LIN {X 0,Y 471.276,Z 351.121,A -85,B 0,C 180,E1 -7520.71,E2 -7520.71} C_VEL
LIN {X 0,Y 472.038,Z 338.499,A -85,B 0,C 180,E1 -7521.712,E2 -7521.712} C_VEL
LIN {X 0,Y 472.825,Z 324.903,A -85,B 0,C 180,E1 -7522.589,E2 -7522.589} C_VEL
LIN {X 0,Y 473.432,Z 311.439,A -85,B 0,C 180,E1 -7523.284,E2 -7523.284} C_VEL
LIN {X 0,Y 473.938,Z 296.086,A -85,B 0,C 180,E1 -7523.884,E2 -7523.884} C_VEL
LIN {X 0,Y 469.116,Z 281.186,A -85,B 0,C 180,E1 -7524.542,E2 -7524.542} C_VEL
LIN {X 0,Y 466.998,Z 274.89,A -85,B 0,C 180,E1 -7524.795,E2 -7524.795} C_VEL
LIN {X 0,Y 467.098,Z 272.572,A -85,B 0,C 180,E1 -7527.412,E2 -7527.412} C_VEL
LIN {X 0,Y 467.145,Z 270.085,A -85,B 0,C 180,E1 -7530.235,E2 -7530.235} C_VEL
LIN {X 0,Y 467.191,Z 267.524,A -85,B 0,C 180,E1 -7533.175,E2 -7533.175} C_VEL
LIN {X 0,Y 467.265,Z 265.036,A -85,B 0,C 180,E1 -7536.041,E2 -7536.041} C_VEL
LIN {X 0,Y 467.335,Z 262.608,A -85,B 0,C 180,E1 -7538.844,E2 -7538.844} C_VEL
LIN {X 0,Y 467.354,Z 261.899,A -85,B 0,C 180,E1 -7539.766,E2 -7539.766} C_VEL
LIN {X 0,Y 467.561,Z 261.875,A -85,B 0,C 180,E1 -7542.506,E2 -7542.506} C_VEL
LIN {X 0,Y 467.599,Z 261.867,A -85,B 0,C 180,E1 -7545.197,E2 -7545.197} C_VEL
LIN {X 0,Y 467.649,Z 261.86,A -85,B 0,C 180,E1 -7547.855,E2 -7547.855} C_VEL
LIN {X 0,Y 467.676,Z 261.856,A -85,B 0,C 180,E1 -7551.358,E2 -7551.358} C_VEL
LIN {X 0,Y 467.739,Z 261.849,A -85,B 0,C 180,E1 -7553.964,E2 -7553.964} C_VEL
LIN {X 0,Y 467.856,Z 261.833,A -85,B 0,C 180,E1 -7557.418,E2 -7557.418} C_VEL
LIN {X 0,Y 467.878,Z 261.829,A -85,B 0,C 180,E1 -7560.001,E2 -7560.001} C_VEL
LIN {X 0,Y 467.856,Z 261.835,A -85,B 0,C 180,E1 -7562.584,E2 -7562.584} C_VEL
LIN {X 0,Y 467.741,Z 261.846,A -85,B 0,C 180,E1 -7566.038,E2 -7566.038} C_VEL
LIN {X 0,Y 467.679,Z 261.855,A -85,B 0,C 180,E1 -7568.644,E2 -7568.644} C_VEL
LIN {X 0,Y 467.653,Z 261.859,A -85,B 0,C 180,E1 -7572.146,E2 -7572.146} C_VEL
LIN {X 0,Y 467.636,Z 261.86,A -85,B 0,C 180,E1 -7575.696,E2 -7575.696} C_VEL
LIN {X 0,Y 467.615,Z 261.863,A -85,B 0,C 180,E1 -7578.766,E2 -7578.766} C_VEL
LIN {X 0,Y 467.579,Z 261.868,A -85,B 0,C 180,E1 -7581.269,E2 -7581.269} C_VEL
LIN {X 0,Y 467.571,Z 261.869,A -85,B 0,C 180,E1 -7583.944,E2 -7583.944} C_VEL
LIN {X 0,Y 467.626,Z 261.863,A -85,B 0,C 180,E1 -7586.8,E2 -7586.8} C_VEL
LIN {X 0,Y 467.552,Z 261.875,A -85,B 0,C 180,E1 -7589.739,E2 -7589.739} C_VEL
LIN {X 0,Y 467.581,Z 261.872,A -85,B 0,C 180,E1 -7592.759,E2 -7592.759} C_VEL
LIN {X 0,Y 467.551,Z 261.878,A -85,B 0,C 180,E1 -7595.89,E2 -7595.89} C_VEL
LIN {X 0,Y 467.581,Z 261.871,A -85,B 0,C 180,E1 -7599.145,E2 -7599.145} C_VEL
LIN {X 0,Y 467.594,Z 262,A -85,B 0,C 180,E1 -7601.978,E2 -7601.978} C_VEL
LIN {X 0,Y 468.651,Z 267.711,A -85,B 0,C 180,E1 -7605.186,E2 -7605.186} C_VEL
LIN {X 0,Y 469.319,Z 271.579,A -85,B 0,C 180,E1 -7607.204,E2 -7607.204} C_VEL
LIN {X 0,Y 469.458,Z 275.977,A -85,B 0,C 180,E1 -7609.34,E2 -7609.34} C_VEL
LIN {X 0,Y 469.141,Z 282.253,A -85,B 0,C 180,E1 -7612.107,E2 -7612.107} C_VEL
LIN {X 0,Y 468.696,Z 290.547,A -85,B 0,C 180,E1 -7615.56,E2 -7615.56} C_VEL
LIN {X 0,Y 468.411,Z 297.548,A -85,B 0,C 180,E1 -7618.323,E2 -7618.323} C_VEL
LIN {X 0,Y 468.186,Z 305.313,A -85,B 0,C 180,E1 -7621.292,E2 -7621.292} C_VEL
LIN {X 0,Y 467.915,Z 313.672,A -85,B 0,C 180,E1 -7624.315,E2 -7624.315} C_VEL
LIN {X 0,Y 467.634,Z 322.474,A -85,B 0,C 180,E1 -7627.466,E2 -7627.466} C_VEL
LIN {X 0,Y 467.569,Z 324.53,A -85,B 0,C 180,E1 -7628.201,E2 -7628.201} C_VEL
LIN {X 0,Y 472.227,Z 343.185,A -85,B 0,C 180,E1 -7628.827,E2 -7628.827} C_VEL
LIN {X 0,Y 473.825,Z 350.535,A -85,B 0,C 180,E1 -7629.124,E2 -7629.124} C_VEL
LIN {X 0,Y 473.197,Z 365.272,A -85,B 0,C 180,E1 -7629.681,E2 -7629.681} C_VEL
LIN {X 0,Y 472.446,Z 380.48,A -85,B 0,C 180,E1 -7630.446,E2 -7630.446} C_VEL
LIN {X 0,Y 471.604,Z 394.063,A -85,B 0,C 180,E1 -7631.314,E2 -7631.314} C_VEL
LIN {X 0,Y 470.728,Z 407.908,A -85,B 0,C 180,E1 -7632.403,E2 -7632.403} C_VEL
LIN {X 0,Y 469.94,Z 420.362,A -85,B 0,C 180,E1 -7633.604,E2 -7633.604} C_VEL
LIN {X 0,Y 469.159,Z 430.752,A -85,B 0,C 180,E1 -7634.803,E2 -7634.803} C_VEL
LIN {X 0,Y 468.478,Z 440.392,A -85,B 0,C 180,E1 -7636.112,E2 -7636.112} C_VEL
LIN {X 0,Y 467.823,Z 449.354,A -85,B 0,C 180,E1 -7637.55,E2 -7637.55} C_VEL
LIN {X 0,Y 467.513,Z 457.737,A -85,B 0,C 180,E1 -7639.17,E2 -7639.17} C_VEL
LIN {X 0,Y 467.072,Z 465.091,A -85,B 0,C 180,E1 -7640.91,E2 -7640.91} C_VEL
LIN {X 0,Y 466.831,Z 470.922,A -85,B 0,C 180,E1 -7642.649,E2 -7642.649} C_VEL
LIN {X 0,Y 466.777,Z 474.387,A -85,B 0,C 180,E1 -7643.951,E2 -7643.951} C_VEL
LIN {X 0,Y 466.62,Z 477.888,A -85,B 0,C 180,E1 -7645.682,E2 -7645.682} C_VEL
LIN {X 0,Y 466.639,Z 480.189,A -85,B 0,C 180,E1 -7647.411,E2 -7647.411} C_VEL
LIN {X 0,Y 466.587,Z 481.348,A -85,B 0,C 180,E1 -7649.138,E2 -7649.138} C_VEL
LIN {X 0,Y 466.587,Z 481.347,A -85,B 0,C 180,E1 -7650.864,E2 -7650.864} C_VEL
LIN {X 0,Y 466.639,Z 480.185,A -85,B 0,C 180,E1 -7652.59,E2 -7652.59} C_VEL
LIN {X 0,Y 466.62,Z 477.881,A -85,B 0,C 180,E1 -7654.319,E2 -7654.319} C_VEL
LIN {X 0,Y 466.751,Z 474.385,A -85,B 0,C 180,E1 -7656.051,E2 -7656.051} C_VEL
LIN {X 0,Y 466.891,Z 469.607,A -85,B 0,C 180,E1 -7657.787,E2 -7657.787} C_VEL
LIN {X 0,Y 467.139,Z 463.417,A -85,B 0,C 180,E1 -7659.526,E2 -7659.526} C_VEL
LIN {X 0,Y 467.628,Z 455.639,A -85,B 0,C 180,E1 -7661.267,E2 -7661.267} C_VEL
LIN {X 0,Y 468.038,Z 447.109,A -85,B 0,C 180,E1 -7662.838,E2 -7662.838} C_VEL
LIN {X 0,Y 468.746,Z 437.387,A -85,B 0,C 180,E1 -7664.324,E2 -7664.324} C_VEL
LIN {X 0,Y 469.354,Z 427.179,A -85,B 0,C 180,E1 -7665.637,E2 -7665.637} C_VEL
LIN {X 0,Y 470.255,Z 414.818,A -85,B 0,C 180,E1 -7666.964,E2 -7666.964} C_VEL
LIN {X 0,Y 471.111,Z 401.347,A -85,B 0,C 180,E1 -7668.145,E2 -7668.145} C_VEL
LIN {X 0,Y 471.975,Z 387.646,A -85,B 0,C 180,E1 -7669.123,E2 -7669.123} C_VEL
LIN {X 0,Y 472.81,Z 373.473,A -85,B 0,C 180,E1 -7669.935,E2 -7669.935} C_VEL
LIN {X 0,Y 473.538,Z 357.964,A -85,B 0,C 180,E1 -7670.619,E2 -7670.619} C_VEL
LIN {X 0,Y 473.65,Z 349.449,A -85,B 0,C 180,E1 -7670.92,E2 -7670.92} C_VEL
LIN {X 0,Y 469.919,Z 334.013,A -85,B 0,C 180,E1 -7671.505,E2 -7671.505} C_VEL
LIN {X 0,Y 467.609,Z 324.753,A -85,B 0,C 180,E1 -7671.797,E2 -7671.797} C_VEL
LIN {X 0,Y 467.901,Z 315.127,A -85,B 0,C 180,E1 -7675.278,E2 -7675.278} C_VEL
LIN {X 0,Y 468.225,Z 305.789,A -85,B 0,C 180,E1 -7678.707,E2 -7678.707} C_VEL
LIN {X 0,Y 468.466,Z 298.067,A -85,B 0,C 180,E1 -7681.674,E2 -7681.674} C_VEL
LIN {X 0,Y 468.842,Z 290.541,A -85,B 0,C 180,E1 -7684.725,E2 -7684.725} C_VEL
LIN {X 0,Y 469.25,Z 282.979,A -85,B 0,C 180,E1 -7687.884,E2 -7687.884} C_VEL
LIN {X 0,Y 469.561,Z 276.677,A -85,B 0,C 180,E1 -7690.664,E2 -7690.664} C_VEL
LIN {X 0,Y 469.383,Z 272.101,A -85,B 0,C 180,E1 -7692.805,E2 -7692.805} C_VEL
LIN {X 0,Y 468.589,Z 267.36,A -85,B 0,C 180,E1 -7695.177,E2 -7695.177} C_VEL
LIN {X 0,Y 467.58,Z 261.869,A -85,B 0,C 180,E1 -7698.165,E2 -7698.165} C_VEL
LIN {X 0,Y 467.567,Z 261.87,A -85,B 0,C 180,E1 -7701.409,E2 -7701.409} C_VEL
LIN {X 0,Y 467.564,Z 261.869,A -85,B 0,C 180,E1 -7704.261,E2 -7704.261} C_VEL
LIN {X 0,Y 467.585,Z 261.867,A -85,B 0,C 180,E1 -7707.321,E2 -7707.321} C_VEL
LIN {X 0,Y 467.574,Z 261.869,A -85,B 0,C 180,E1 -7710.667,E2 -7710.667} C_VEL
LIN {X 0,Y 467.622,Z 261.862,A -85,B 0,C 180,E1 -7713.199,E2 -7713.199} C_VEL
LIN {X 0,Y 467.598,Z 261.867,A -85,B 0,C 180,E1 -7716.468,E2 -7716.468} C_VEL
LIN {X 0,Y 467.629,Z 261.859,A -85,B 0,C 180,E1 -7719.777,E2 -7719.777} C_VEL
LIN {X 0,Y 467.615,Z 261.865,A -85,B 0,C 180,E1 -7722.506,E2 -7722.506} C_VEL
LIN {X 0,Y 467.611,Z 261.864,A -85,B 0,C 180,E1 -7725.196,E2 -7725.196} C_VEL
LIN {X 0,Y 467.661,Z 261.857,A -85,B 0,C 180,E1 -7727.854,E2 -7727.854} C_VEL
LIN {X 0,Y 467.685,Z 261.853,A -85,B 0,C 180,E1 -7731.356,E2 -7731.356} C_VEL
LIN {X 0,Y 467.726,Z 261.849,A -85,B 0,C 180,E1 -7733.962,E2 -7733.962} C_VEL
LIN {X 0,Y 467.864,Z 261.83,A -85,B 0,C 180,E1 -7737.416,E2 -7737.416} C_VEL
LIN {X 0,Y 467.887,Z 261.829,A -85,B 0,C 180,E1 -7739.999,E2 -7739.999} C_VEL
LIN {X 0,Y 467.862,Z 261.833,A -85,B 0,C 180,E1 -7742.582,E2 -7742.582} C_VEL
LIN {X 0,Y 467.746,Z 261.847,A -85,B 0,C 180,E1 -7746.036,E2 -7746.036} C_VEL
LIN {X 0,Y 467.684,Z 261.855,A -85,B 0,C 180,E1 -7748.642,E2 -7748.642} C_VEL
LIN {X 0,Y 467.658,Z 261.859,A -85,B 0,C 180,E1 -7752.144,E2 -7752.144} C_VEL
LIN {X 0,Y 467.641,Z 261.859,A -85,B 0,C 180,E1 -7755.694,E2 -7755.694} C_VEL
LIN {X 0,Y 467.618,Z 261.863,A -85,B 0,C 180,E1 -7758.763,E2 -7758.763} C_VEL
LIN {X 0,Y 467.581,Z 261.866,A -85,B 0,C 180,E1 -7761.267,E2 -7761.267} C_VEL
LIN {X 0,Y 467.573,Z 261.869,A -85,B 0,C 180,E1 -7763.942,E2 -7763.942} C_VEL
LIN {X 0,Y 467.616,Z 261.862,A -85,B 0,C 180,E1 -7766.799,E2 -7766.799} C_VEL
LIN {X 0,Y 467.553,Z 261.873,A -85,B 0,C 180,E1 -7769.737,E2 -7769.737} C_VEL
LIN {X 0,Y 467.581,Z 261.866,A -85,B 0,C 180,E1 -7772.757,E2 -7772.757} C_VEL
LIN {X 0,Y 467.554,Z 261.873,A -85,B 0,C 180,E1 -7775.888,E2 -7775.888} C_VEL
LIN {X 0,Y 467.579,Z 261.867,A -85,B 0,C 180,E1 -7779.143,E2 -7779.143} C_VEL
LIN {X 0,Y 467.582,Z 261.867,A -85,B 0,C 180,E1 -7782.566,E2 -7782.566} C_VEL
LIN {X 0,Y 467.566,Z 261.868,A -85,B 0,C 180,E1 -7785.052,E2 -7785.052} C_VEL
LIN {X 0,Y 467.619,Z 261.864,A -85,B 0,C 180,E1 -7787.443,E2 -7787.443} C_VEL
LIN {X 0,Y 467.594,Z 261.864,A -85,B 0,C 180,E1 -7790.856,E2 -7790.856} C_VEL
LIN {X 0,Y 467.556,Z 261.871,A -85,B 0,C 180,E1 -7794.259,E2 -7794.259} C_VEL
LIN {X 0,Y 467.575,Z 261.869,A -85,B 0,C 180,E1 -7797.32,E2 -7797.32} C_VEL
LIN {X 0,Y 467.57,Z 261.867,A -85,B 0,C 180,E1 -7800.664,E2 -7800.664} C_VEL
LIN {X 0,Y 467.62,Z 261.864,A -85,B 0,C 180,E1 -7803.199,E2 -7803.199} C_VEL
LIN {X 0,Y 467.584,Z 261.865,A -85,B 0,C 180,E1 -7806.467,E2 -7806.467} C_VEL
LIN {X 0,Y 467.615,Z 261.864,A -85,B 0,C 180,E1 -7809.776,E2 -7809.776} C_VEL
LIN {X 0,Y 467.6,Z 261.864,A -85,B 0,C 180,E1 -7812.506,E2 -7812.506} C_VEL
LIN {X 0,Y 467.59,Z 261.866,A -85,B 0,C 180,E1 -7815.418,E2 -7815.418} C_VEL
LIN {X 0,Y 466.921,Z 261.949,A -85,B 0,C 180,E1 -7816.137,E2 -7816.137} C_VEL
LIN {X 0,Y 464.086,Z 262.304,A -85,B 0,C 180,E1 -7817.306,E2 -7817.306} C_VEL
LIN {X 0,Y 461.692,Z 262.599,A -85,B 0,C 180,E1 -7818.248,E2 -7818.248} C_VEL
LIN {X 0,Y 460.665,Z 262.73,A -85,B 0,C 180,E1 -7818.976,E2 -7818.976} C_VEL
LIN {X 0,Y 460.581,Z 262.739,A -85,B 0,C 180,E1 -7819.223,E2 -7819.223} C_VEL
LIN {X 0,Y 460.709,Z 262.721,A -85,B 0,C 180,E1 -7822.537,E2 -7822.537} C_VEL
LIN {X 0,Y 460.668,Z 262.727,A -85,B 0,C 180,E1 -7824.747,E2 -7824.747} C_VEL
LIN {X 0,Y 460.337,Z 262.772,A -85,B 0,C 180,E1 -7828.25,E2 -7828.25} C_VEL
LIN {X 0,Y 460.531,Z 263.298,A -85,B 0,C 180,E1 -7829.125,E2 -7829.125} C_VEL
LIN {X 0,Y 460.006,Z 265.723,A -85,B 0,C 180,E1 -7831.75,E2 -7831.75} C_VEL
LIN {X 0,Y 460.14,Z 268.114,A -85,B 0,C 180,E1 -7834.379,E2 -7834.379} C_VEL
LIN {X 0,Y 460.034,Z 270.553,A -85,B 0,C 180,E1 -7837.019,E2 -7837.019} C_VEL
LIN {X 0,Y 459.895,Z 273.884,A -85,B 0,C 180,E1 -7840.566,E2 -7840.566} C_VEL
LIN {X 0,Y 459.941,Z 274.351,A -85,B 0,C 180,E1 -7840.983,E2 -7840.983} C_VEL
LIN {X 0,Y 464.985,Z 289.981,A -85,B 0,C 180,E1 -7841.608,E2 -7841.608} C_VEL
LIN {X 0,Y 467.218,Z 298.137,A -85,B 0,C 180,E1 -7841.99,E2 -7841.99} C_VEL
LIN {X 0,Y 466.607,Z 312.198,A -85,B 0,C 180,E1 -7842.559,E2 -7842.559} C_VEL
LIN {X 0,Y 465.902,Z 326.161,A -85,B 0,C 180,E1 -7843.299,E2 -7843.299} C_VEL
LIN {X 0,Y 465.029,Z 340.681,A -85,B 0,C 180,E1 -7844.276,E2 -7844.276} C_VEL
LIN {X 0,Y 464.213,Z 353.744,A -85,B 0,C 180,E1 -7845.363,E2 -7845.363} C_VEL
LIN {X 0,Y 463.314,Z 366.347,A -85,B 0,C 180,E1 -7846.637,E2 -7846.637} C_VEL
LIN {X 0,Y 462.534,Z 376.968,A -85,B 0,C 180,E1 -7847.919,E2 -7847.919} C_VEL
LIN {X 0,Y 461.764,Z 386.826,A -85,B 0,C 180,E1 -7849.334,E2 -7849.334} C_VEL
LIN {X 0,Y 461.099,Z 396.378,A -85,B 0,C 180,E1 -7850.988,E2 -7850.988} C_VEL
LIN {X 0,Y 460.593,Z 404.304,A -85,B 0,C 180,E1 -7852.66,E2 -7852.66} C_VEL
LIN {X 0,Y 460.154,Z 410.823,A -85,B 0,C 180,E1 -7854.353,E2 -7854.353} C_VEL
LIN {X 0,Y 459.972,Z 414.87,A -85,B 0,C 180,E1 -7855.651,E2 -7855.651} C_VEL
LIN {X 0,Y 459.816,Z 419.011,A -85,B 0,C 180,E1 -7857.292,E2 -7857.292} C_VEL
LIN {X 0,Y 459.575,Z 422.573,A -85,B 0,C 180,E1 -7859.297,E2 -7859.297} C_VEL
LIN {X 0,Y 459.501,Z 424.629,A -85,B 0,C 180,E1 -7861.333,E2 -7861.333} C_VEL
LIN {X 0,Y 459.49,Z 425.161,A -85,B 0,C 180,E1 -7862.732,E2 -7862.732} C_VEL
LIN {X 0,Y 459.493,Z 424.833,A -85,B 0,C 180,E1 -7864.465,E2 -7864.465} C_VEL
LIN {X 0,Y 459.532,Z 423.811,A -85,B 0,C 180,E1 -7865.851,E2 -7865.851} C_VEL
LIN {X 0,Y 459.65,Z 421.28,A -85,B 0,C 180,E1 -7867.704,E2 -7867.704} C_VEL
LIN {X 0,Y 459.865,Z 417.877,A -85,B 0,C 180,E1 -7869.362,E2 -7869.362} C_VEL
LIN {X 0,Y 460.082,Z 413.253,A -85,B 0,C 180,E1 -7871.059,E2 -7871.059} C_VEL
LIN {X 0,Y 460.459,Z 406.789,A -85,B 0,C 180,E1 -7872.895,E2 -7872.895} C_VEL
LIN {X 0,Y 460.954,Z 399.585,A -85,B 0,C 180,E1 -7874.534,E2 -7874.534} C_VEL
LIN {X 0,Y 461.498,Z 391.742,A -85,B 0,C 180,E1 -7876.017,E2 -7876.017} C_VEL
LIN {X 0,Y 462.198,Z 382.244,A -85,B 0,C 180,E1 -7877.515,E2 -7877.515} C_VEL
LIN {X 0,Y 462.97,Z 372.017,A -85,B 0,C 180,E1 -7878.865,E2 -7878.865} C_VEL
LIN {X 0,Y 463.912,Z 359.837,A -85,B 0,C 180,E1 -7880.205,E2 -7880.205} C_VEL
LIN {X 0,Y 464.783,Z 348.128,A -85,B 0,C 180,E1 -7881.273,E2 -7881.273} C_VEL
LIN {X 0,Y 465.468,Z 336.276,A -85,B 0,C 180,E1 -7882.182,E2 -7882.182} C_VEL
LIN {X 0,Y 466.295,Z 322.92,A -85,B 0,C 180,E1 -7883.016,E2 -7883.016} C_VEL
LIN {X 0,Y 466.924,Z 308.685,A -85,B 0,C 180,E1 -7883.723,E2 -7883.723} C_VEL
LIN {X 0,Y 467.169,Z 297.157,A -85,B 0,C 180,E1 -7884.18,E2 -7884.18} C_VEL
LIN {X 0,Y 462.212,Z 282.074,A -85,B 0,C 180,E1 -7884.873,E2 -7884.873} C_VEL
LIN {X 0,Y 459.948,Z 275.393,A -85,B 0,C 180,E1 -7885.142,E2 -7885.142} C_VEL
LIN {X 0,Y 460.034,Z 273.151,A -85,B 0,C 180,E1 -7887.678,E2 -7887.678} C_VEL
LIN {X 0,Y 460.117,Z 270.488,A -85,B 0,C 180,E1 -7890.741,E2 -7890.741} C_VEL
LIN {X 0,Y 460.166,Z 267.939,A -85,B 0,C 180,E1 -7893.712,E2 -7893.712} C_VEL
LIN {X 0,Y 460.287,Z 265.428,A -85,B 0,C 180,E1 -7896.611,E2 -7896.611} C_VEL
LIN {X 0,Y 460.288,Z 263.03,A -85,B 0,C 180,E1 -7899.442,E2 -7899.442} C_VEL
LIN {X 0,Y 460.483,Z 262.755,A -85,B 0,C 180,E1 -7901.308,E2 -7901.308} C_VEL
LIN {X 0,Y 460.596,Z 262.74,A -85,B 0,C 180,E1 -7904.06,E2 -7904.06} C_VEL
LIN {X 0,Y 460.602,Z 262.739,A -85,B 0,C 180,E1 -7907.667,E2 -7907.667} C_VEL
LIN {X 0,Y 460.623,Z 262.735,A -85,B 0,C 180,E1 -7911.225,E2 -7911.225} C_VEL
LIN {X 0,Y 460.705,Z 262.725,A -85,B 0,C 180,E1 -7913.871,E2 -7913.871} C_VEL
LIN {X 0,Y 460.821,Z 262.71,A -85,B 0,C 180,E1 -7917.379,E2 -7917.379} C_VEL
LIN {X 0,Y 460.849,Z 262.705,A -85,B 0,C 180,E1 -7920.001,E2 -7920.001} C_VEL
LIN {X 0,Y 460.821,Z 262.711,A -85,B 0,C 180,E1 -7922.623,E2 -7922.623} C_VEL
LIN {X 0,Y 460.707,Z 262.722,A -85,B 0,C 180,E1 -7926.131,E2 -7926.131} C_VEL
LIN {X 0,Y 460.626,Z 262.733,A -85,B 0,C 180,E1 -7928.777,E2 -7928.777} C_VEL
LIN {X 0,Y 460.61,Z 262.735,A -85,B 0,C 180,E1 -7932.446,E2 -7932.446} C_VEL
LIN {X 0,Y 460.597,Z 262.737,A -85,B 0,C 180,E1 -7935.998,E2 -7935.998} C_VEL
LIN {X 0,Y 460.568,Z 262.74,A -85,B 0,C 180,E1 -7938.903,E2 -7938.903} C_VEL
LIN {X 0,Y 460.513,Z 262.747,A -85,B 0,C 180,E1 -7941.486,E2 -7941.486} C_VEL
LIN {X 0,Y 460.54,Z 262.745,A -85,B 0,C 180,E1 -7944.333,E2 -7944.333} C_VEL
LIN {X 0,Y 460.582,Z 262.738,A -85,B 0,C 180,E1 -7947.244,E2 -7947.244} C_VEL
LIN {X 0,Y 460.508,Z 262.752,A -85,B 0,C 180,E1 -7950.241,E2 -7950.241} C_VEL
LIN {X 0,Y 460.527,Z 262.752,A -85,B 0,C 180,E1 -7953.326,E2 -7953.326} C_VEL
LIN {X 0,Y 460.474,Z 262.758,A -85,B 0,C 180,E1 -7956.53,E2 -7956.53} C_VEL
LIN {X 0,Y 460.531,Z 262.75,A -85,B 0,C 180,E1 -7959.863,E2 -7959.863} C_VEL
LIN {X 0,Y 460.565,Z 262.934,A -85,B 0,C 180,E1 -7961.608,E2 -7961.608} C_VEL
LIN {X 0,Y 461.648,Z 268.875,A -85,B 0,C 180,E1 -7965.024,E2 -7965.024} C_VEL
LIN {X 0,Y 462.414,Z 273.472,A -85,B 0,C 180,E1 -7967.459,E2 -7967.459} C_VEL
LIN {X 0,Y 462.483,Z 277.628,A -85,B 0,C 180,E1 -7969.448,E2 -7969.448} C_VEL
LIN {X 0,Y 462.087,Z 284.474,A -85,B 0,C 180,E1 -7972.529,E2 -7972.529} C_VEL
LIN {X 0,Y 461.643,Z 292.04,A -85,B 0,C 180,E1 -7975.718,E2 -7975.718} C_VEL
LIN {X 0,Y 461.353,Z 299.097,A -85,B 0,C 180,E1 -7978.548,E2 -7978.548} C_VEL
LIN {X 0,Y 461.131,Z 306.199,A -85,B 0,C 180,E1 -7981.31,E2 -7981.31} C_VEL
LIN {X 0,Y 460.791,Z 315.429,A -85,B 0,C 180,E1 -7984.72,E2 -7984.72} C_VEL
LIN {X 0,Y 460.527,Z 324.052,A -85,B 0,C 180,E1 -7987.862,E2 -7987.862} C_VEL
LIN {X 0,Y 463.894,Z 337.773,A -85,B 0,C 180,E1 -7988.303,E2 -7988.303} C_VEL
LIN {X 0,Y 467.097,Z 351.682,A -85,B 0,C 180,E1 -7988.868,E2 -7988.868} C_VEL
LIN {X 0,Y 466.485,Z 365.479,A -85,B 0,C 180,E1 -7989.407,E2 -7989.407} C_VEL
LIN {X 0,Y 465.695,Z 379.972,A -85,B 0,C 180,E1 -7990.151,E2 -7990.151} C_VEL
LIN {X 0,Y 464.811,Z 393.557,A -85,B 0,C 180,E1 -7991.03,E2 -7991.03} C_VEL
LIN {X 0,Y 463.877,Z 407.406,A -85,B 0,C 180,E1 -7992.134,E2 -7992.134} C_VEL
LIN {X 0,Y 463.049,Z 419.961,A -85,B 0,C 180,E1 -7993.353,E2 -7993.353} C_VEL
LIN {X 0,Y 462.101,Z 432.278,A -85,B 0,C 180,E1 -7994.791,E2 -7994.791} C_VEL
LIN {X 0,Y 461.31,Z 443.239,A -85,B 0,C 180,E1 -7996.342,E2 -7996.342} C_VEL
LIN {X 0,Y 460.686,Z 452.3,A -85,B 0,C 180,E1 -7997.892,E2 -7997.892} C_VEL
LIN {X 0,Y 460.293,Z 459.752,A -85,B 0,C 180,E1 -7999.443,E2 -7999.443} C_VEL
LIN {X 0,Y 459.94,Z 466.702,A -85,B 0,C 180,E1 -8001.211,E2 -8001.211} C_VEL
LIN {X 0,Y 459.737,Z 472.164,A -85,B 0,C 180,E1 -8002.976,E2 -8002.976} C_VEL
LIN {X 0,Y 459.638,Z 476.291,A -85,B 0,C 180,E1 -8004.737,E2 -8004.737} C_VEL
LIN {X 0,Y 459.54,Z 479.184,A -85,B 0,C 180,E1 -8006.493,E2 -8006.493} C_VEL
LIN {X 0,Y 459.514,Z 480.909,A -85,B 0,C 180,E1 -8008.248,E2 -8008.248} C_VEL
LIN {X 0,Y 459.472,Z 481.5,A -85,B 0,C 180,E1 -8010.001,E2 -8010.001} C_VEL
LIN {X 0,Y 459.514,Z 480.906,A -85,B 0,C 180,E1 -8011.753,E2 -8011.753} C_VEL
LIN {X 0,Y 459.541,Z 479.178,A -85,B 0,C 180,E1 -8013.508,E2 -8013.508} C_VEL
LIN {X 0,Y 459.633,Z 476.286,A -85,B 0,C 180,E1 -8015.264,E2 -8015.264} C_VEL
LIN {X 0,Y 459.733,Z 472.164,A -85,B 0,C 180,E1 -8017.025,E2 -8017.025} C_VEL
LIN {X 0,Y 459.942,Z 466.698,A -85,B 0,C 180,E1 -8018.79,E2 -8018.79} C_VEL
LIN {X 0,Y 460.294,Z 459.74,A -85,B 0,C 180,E1 -8020.558,E2 -8020.558} C_VEL
LIN {X 0,Y 460.719,Z 452.29,A -85,B 0,C 180,E1 -8022.108,E2 -8022.108} C_VEL
LIN {X 0,Y 461.307,Z 443.235,A -85,B 0,C 180,E1 -8023.66,E2 -8023.66} C_VEL
LIN {X 0,Y 462.103,Z 432.289,A -85,B 0,C 180,E1 -8025.21,E2 -8025.21} C_VEL
LIN {X 0,Y 462.959,Z 421.028,A -85,B 0,C 180,E1 -8026.538,E2 -8026.538} C_VEL
LIN {X 0,Y 463.825,Z 408.701,A -85,B 0,C 180,E1 -8027.755,E2 -8027.755} C_VEL
LIN {X 0,Y 464.746,Z 395.164,A -85,B 0,C 180,E1 -8028.859,E2 -8028.859} C_VEL
LIN {X 0,Y 465.525,Z 381.879,A -85,B 0,C 180,E1 -8029.743,E2 -8029.743} C_VEL
LIN {X 0,Y 466.411,Z 367.456,A -85,B 0,C 180,E1 -8030.505,E2 -8030.505} C_VEL
LIN {X 0,Y 467.07,Z 352.57,A -85,B 0,C 180,E1 -8031.106,E2 -8031.106} C_VEL
LIN {X 0,Y 466.079,Z 346.767,A -85,B 0,C 180,E1 -8031.346,E2 -8031.346} C_VEL
LIN {X 0,Y 462.031,Z 330.784,A -85,B 0,C 180,E1 -8031.945,E2 -8031.945} C_VEL
LIN {X 0,Y 460.555,Z 324.34,A -85,B 0,C 180,E1 -8032.144,E2 -8032.144} C_VEL
LIN {X 0,Y 460.843,Z 315.932,A -85,B 0,C 180,E1 -8035.278,E2 -8035.278} C_VEL
LIN {X 0,Y 461.173,Z 306.783,A -85,B 0,C 180,E1 -8038.689,E2 -8038.689} C_VEL
LIN {X 0,Y 461.444,Z 299.654,A -85,B 0,C 180,E1 -8041.47,E2 -8041.47} C_VEL
LIN {X 0,Y 461.756,Z 292.774,A -85,B 0,C 180,E1 -8044.274,E2 -8044.274} C_VEL
LIN {X 0,Y 462.186,Z 285.218,A -85,B 0,C 180,E1 -8047.463,E2 -8047.463} C_VEL
LIN {X 0,Y 462.533,Z 279.258,A -85,B 0,C 180,E1 -8050.11,E2 -8050.11} C_VEL
LIN {X 0,Y 462.591,Z 275.286,A -85,B 0,C 180,E1 -8051.95,E2 -8051.95} C_VEL
LIN {X 0,Y 461.927,Z 270.334,A -85,B 0,C 180,E1 -8054.417,E2 -8054.417} C_VEL
LIN {X 0,Y 460.764,Z 263.934,A -85,B 0,C 180,E1 -8057.845,E2 -8057.845} C_VEL
LIN {X 0,Y 460.559,Z 262.743,A -85,B 0,C 180,E1 -8058.58,E2 -8058.58} C_VEL
LIN {X 0,Y 460.531,Z 262.746,A -85,B 0,C 180,E1 -8061.267,E2 -8061.267} C_VEL
LIN {X 0,Y 460.514,Z 262.749,A -85,B 0,C 180,E1 -8064.554,E2 -8064.554} C_VEL
LIN {X 0,Y 460.535,Z 262.747,A -85,B 0,C 180,E1 -8067.715,E2 -8067.715} C_VEL
LIN {X 0,Y 460.544,Z 262.746,A -85,B 0,C 180,E1 -8070.769,E2 -8070.769} C_VEL
LIN {X 0,Y 460.569,Z 262.739,A -85,B 0,C 180,E1 -8073.734,E2 -8073.734} C_VEL
LIN {X 0,Y 460.552,Z 262.744,A -85,B 0,C 180,E1 -8076.624,E2 -8076.624} C_VEL
LIN {X 0,Y 460.557,Z 262.74,A -85,B 0,C 180,E1 -8079.452,E2 -8079.452} C_VEL
LIN {X 0,Y 460.565,Z 262.741,A -85,B 0,C 180,E1 -8082.23,E2 -8082.23} C_VEL
LIN {X 0,Y 460.571,Z 262.741,A -85,B 0,C 180,E1 -8084.964,E2 -8084.964} C_VEL
LIN {X 0,Y 460.615,Z 262.737,A -85,B 0,C 180,E1 -8088.559,E2 -8088.559} C_VEL
LIN {X 0,Y 460.672,Z 262.729,A -85,B 0,C 180,E1 -8092.107,E2 -8092.107} C_VEL
LIN {X 0,Y 460.694,Z 262.727,A -85,B 0,C 180,E1 -8094.747,E2 -8094.747} C_VEL
LIN {X 0,Y 460.805,Z 262.709,A -85,B 0,C 180,E1 -8097.377,E2 -8097.377} C_VEL
LIN {X 0,Y 460.857,Z 262.705,A -85,B 0,C 180,E1 -8099.999,E2 -8099.999} C_VEL
LIN {X 0,Y 460.803,Z 262.713,A -85,B 0,C 180,E1 -8102.622,E2 -8102.622} C_VEL
LIN {X 0,Y 460.712,Z 262.724,A -85,B 0,C 180,E1 -8106.129,E2 -8106.129} C_VEL
LIN {X 0,Y 460.631,Z 262.733,A -85,B 0,C 180,E1 -8108.775,E2 -8108.775} C_VEL
LIN {X 0,Y 460.616,Z 262.737,A -85,B 0,C 180,E1 -8112.444,E2 -8112.444} C_VEL
LIN {X 0,Y 460.602,Z 262.739,A -85,B 0,C 180,E1 -8115.996,E2 -8115.996} C_VEL
LIN {X 0,Y 460.572,Z 262.739,A -85,B 0,C 180,E1 -8118.9,E2 -8118.9} C_VEL
LIN {X 0,Y 460.516,Z 262.747,A -85,B 0,C 180,E1 -8121.484,E2 -8121.484} C_VEL
LIN {X 0,Y 460.543,Z 262.745,A -85,B 0,C 180,E1 -8124.331,E2 -8124.331} C_VEL
LIN {X 0,Y 460.579,Z 262.738,A -85,B 0,C 180,E1 -8127.242,E2 -8127.242} C_VEL
LIN {X 0,Y 460.509,Z 262.75,A -85,B 0,C 180,E1 -8130.239,E2 -8130.239} C_VEL
LIN {X 0,Y 460.527,Z 262.745,A -85,B 0,C 180,E1 -8133.323,E2 -8133.323} C_VEL
LIN {X 0,Y 460.476,Z 262.752,A -85,B 0,C 180,E1 -8136.528,E2 -8136.528} C_VEL
LIN {X 0,Y 460.554,Z 262.745,A -85,B 0,C 180,E1 -8139.858,E2 -8139.858} C_VEL
LIN {X 0,Y 460.512,Z 262.746,A -85,B 0,C 180,E1 -8142.9,E2 -8142.9} C_VEL
LIN {X 0,Y 460.519,Z 262.748,A -85,B 0,C 180,E1 -8145.827,E2 -8145.827} C_VEL
LIN {X 0,Y 460.537,Z 262.742,A -85,B 0,C 180,E1 -8148.989,E2 -8148.989} C_VEL
LIN {X 0,Y 460.533,Z 262.745,A -85,B 0,C 180,E1 -8151.267,E2 -8151.267} C_VEL
LIN {X 0,Y 460.507,Z 262.747,A -85,B 0,C 180,E1 -8154.553,E2 -8154.553} C_VEL
LIN {X 0,Y 460.525,Z 262.748,A -85,B 0,C 180,E1 -8157.715,E2 -8157.715} C_VEL
LIN {X 0,Y 460.539,Z 262.743,A -85,B 0,C 180,E1 -8160.768,E2 -8160.768} C_VEL
LIN {X 0,Y 460.56,Z 262.744,A -85,B 0,C 180,E1 -8163.734,E2 -8163.734} C_VEL
LIN {X 0,Y 460.537,Z 262.742,A -85,B 0,C 180,E1 -8166.623,E2 -8166.623} C_VEL
LIN {X 0,Y 460.543,Z 262.746,A -85,B 0,C 180,E1 -8169.452,E2 -8169.452} C_VEL
LIN {X 0,Y 460.55,Z 262.742,A -85,B 0,C 180,E1 -8172.229,E2 -8172.229} C_VEL
LIN {X 0,Y 460.557,Z 262.742,A -85,B 0,C 180,E1 -8174.964,E2 -8174.964} C_VEL
LIN {X 0,Y 460.619,Z 262.735,A -85,B 0,C 180,E1 -8177.666,E2 -8177.666} C_VEL
LIN {X 0,Y 460.581,Z 262.739,A -85,B 0,C 180,E1 -8179.223,E2 -8179.223} C_VEL
LIN {X 0,Y 459.921,Z 262.826,A -85,B 0,C 180,E1 -8179.953,E2 -8179.953} C_VEL
LIN {X 0,Y 457.1,Z 263.179,A -85,B 0,C 180,E1 -8181.139,E2 -8181.139} C_VEL
LIN {X 0,Y 454.719,Z 263.473,A -85,B 0,C 180,E1 -8182.096,E2 -8182.096} C_VEL
LIN {X 0,Y 453.703,Z 263.596,A -85,B 0,C 180,E1 -8182.835,E2 -8182.835} C_VEL
LIN {X 0,Y 453.624,Z 263.605,A -85,B 0,C 180,E1 -8183.085,E2 -8183.085} C_VEL
LIN {X 0,Y 453.643,Z 263.602,A -85,B 0,C 180,E1 -8184.666,E2 -8184.666} C_VEL
LIN {X 0,Y 453.305,Z 263.648,A -85,B 0,C 180,E1 -8188.222,E2 -8188.222} C_VEL
LIN {X 0,Y 453.494,Z 264.085,A -85,B 0,C 180,E1 -8189.111,E2 -8189.111} C_VEL
LIN {X 0,Y 452.944,Z 266.533,A -85,B 0,C 180,E1 -8191.778,E2 -8191.778} C_VEL
LIN {X 0,Y 453.07,Z 268.943,A -85,B 0,C 180,E1 -8194.448,E2 -8194.448} C_VEL
LIN {X 0,Y 452.969,Z 271.396,A -85,B 0,C 180,E1 -8197.129,E2 -8197.129} C_VEL
LIN {X 0,Y 452.842,Z 274.656,A -85,B 0,C 180,E1 -8200.62,E2 -8200.62} C_VEL
LIN {X 0,Y 458.106,Z 290.711,A -85,B 0,C 180,E1 -8201.287,E2 -8201.287} C_VEL
LIN {X 0,Y 460.53,Z 298.991,A -85,B 0,C 180,E1 -8201.693,E2 -8201.693} C_VEL
LIN {X 0,Y 459.907,Z 313.511,A -85,B 0,C 180,E1 -8202.301,E2 -8202.301} C_VEL
LIN {X 0,Y 459.177,Z 327.205,A -85,B 0,C 180,E1 -8203.047,E2 -8203.047} C_VEL
LIN {X 0,Y 458.328,Z 340.81,A -85,B 0,C 180,E1 -8203.975,E2 -8203.975} C_VEL
LIN {X 0,Y 457.557,Z 353.01,A -85,B 0,C 180,E1 -8204.993,E2 -8204.993} C_VEL
LIN {X 0,Y 456.606,Z 365.057,A -85,B 0,C 180,E1 -8206.198,E2 -8206.198} C_VEL
LIN {X 0,Y 455.743,Z 375.563,A -85,B 0,C 180,E1 -8207.453,E2 -8207.453} C_VEL
LIN {X 0,Y 454.925,Z 385.965,A -85,B 0,C 180,E1 -8208.93,E2 -8208.93} C_VEL
LIN {X 0,Y 454.281,Z 394.464,A -85,B 0,C 180,E1 -8210.37,E2 -8210.37} C_VEL
LIN {X 0,Y 453.698,Z 402.791,A -85,B 0,C 180,E1 -8212.063,E2 -8212.063} C_VEL
LIN {X 0,Y 453.22,Z 409.791,A -85,B 0,C 180,E1 -8213.812,E2 -8213.812} C_VEL
LIN {X 0,Y 452.886,Z 415.891,A -85,B 0,C 180,E1 -8215.753,E2 -8215.753} C_VEL
LIN {X 0,Y 452.754,Z 419.529,A -85,B 0,C 180,E1 -8217.248,E2 -8217.248} C_VEL
LIN {X 0,Y 452.522,Z 422.324,A -85,B 0,C 180,E1 -8218.78,E2 -8218.78} C_VEL
LIN {X 0,Y 452.445,Z 424.734,A -85,B 0,C 180,E1 -8220.836,E2 -8220.836} C_VEL
LIN {X 0,Y 452.393,Z 425.384,A -85,B 0,C 180,E1 -8221.883,E2 -8221.883} C_VEL
LIN {X 0,Y 452.409,Z 425.653,A -85,B 0,C 180,E1 -8222.982,E2 -8222.982} C_VEL
LIN {X 0,Y 452.406,Z 425.229,A -85,B 0,C 180,E1 -8224.582,E2 -8224.582} C_VEL
LIN {X 0,Y 452.462,Z 423.963,A -85,B 0,C 180,E1 -8226.174,E2 -8226.174} C_VEL
LIN {X 0,Y 452.571,Z 421.959,A -85,B 0,C 180,E1 -8227.631,E2 -8227.631} C_VEL
LIN {X 0,Y 452.804,Z 418.191,A -85,B 0,C 180,E1 -8229.52,E2 -8229.52} C_VEL
LIN {X 0,Y 453.067,Z 413.523,A -85,B 0,C 180,E1 -8231.243,E2 -8231.243} C_VEL
LIN {X 0,Y 453.432,Z 407.448,A -85,B 0,C 180,E1 -8232.998,E2 -8232.998} C_VEL
LIN {X 0,Y 453.946,Z 400.641,A -85,B 0,C 180,E1 -8234.59,E2 -8234.59} C_VEL
LIN {X 0,Y 454.563,Z 392.308,A -85,B 0,C 180,E1 -8236.2,E2 -8236.2} C_VEL
LIN {X 0,Y 455.351,Z 382.254,A -85,B 0,C 180,E1 -8237.802,E2 -8237.802} C_VEL
LIN {X 0,Y 456.229,Z 371.723,A -85,B 0,C 180,E1 -8239.199,E2 -8239.199} C_VEL
LIN {X 0,Y 457.122,Z 360.599,A -85,B 0,C 180,E1 -8240.436,E2 -8240.436} C_VEL
LIN {X 0,Y 458.106,Z 347.257,A -85,B 0,C 180,E1 -8241.666,E2 -8241.666} C_VEL
LIN {X 0,Y 458.979,Z 334.303,A -85,B 0,C 180,E1 -8242.643,E2 -8242.643} C_VEL
LIN {X 0,Y 459.813,Z 320.534,A -85,B 0,C 180,E1 -8243.479,E2 -8243.479} C_VEL
LIN {X 0,Y 460.422,Z 306.906,A -85,B 0,C 180,E1 -8244.131,E2 -8244.131} C_VEL
LIN {X 0,Y 460.532,Z 298.755,A -85,B 0,C 180,E1 -8244.457,E2 -8244.457} C_VEL
LIN {X 0,Y 455.833,Z 284.268,A -85,B 0,C 180,E1 -8245.152,E2 -8245.152} C_VEL
LIN {X 0,Y 452.96,Z 276.15,A -85,B 0,C 180,E1 -8245.484,E2 -8245.484} C_VEL
LIN {X 0,Y 452.93,Z 275.84,A -85,B 0,C 180,E1 -8245.561,E2 -8245.561} C_VEL
LIN {X 0,Y 453,Z 273.225,A -85,B 0,C 180,E1 -8248.57,E2 -8248.57} C_VEL
LIN {X 0,Y 453.071,Z 270.892,A -85,B 0,C 180,E1 -8251.259,E2 -8251.259} C_VEL
LIN {X 0,Y 453.174,Z 268.335,A -85,B 0,C 180,E1 -8254.265,E2 -8254.265} C_VEL
LIN {X 0,Y 453.229,Z 265.855,A -85,B 0,C 180,E1 -8257.192,E2 -8257.192} C_VEL
LIN {X 0,Y 453.298,Z 263.65,A -85,B 0,C 180,E1 -8260.058,E2 -8260.058} C_VEL
LIN {X 0,Y 453.472,Z 263.629,A -85,B 0,C 180,E1 -8262.876,E2 -8262.876} C_VEL
LIN {X 0,Y 453.506,Z 263.623,A -85,B 0,C 180,E1 -8265.645,E2 -8265.645} C_VEL
LIN {X 0,Y 453.554,Z 263.615,A -85,B 0,C 180,E1 -8268.38,E2 -8268.38} C_VEL
LIN {X 0,Y 453.646,Z 263.605,A -85,B 0,C 180,E1 -8271.986,E2 -8271.986} C_VEL
LIN {X 0,Y 453.668,Z 263.601,A -85,B 0,C 180,E1 -8274.668,E2 -8274.668} C_VEL
LIN {X 0,Y 453.761,Z 263.589,A -85,B 0,C 180,E1 -8277.338,E2 -8277.338} C_VEL
LIN {X 0,Y 453.819,Z 263.58,A -85,B 0,C 180,E1 -8280.001,E2 -8280.001} C_VEL
LIN {X 0,Y 453.761,Z 263.591,A -85,B 0,C 180,E1 -8282.664,E2 -8282.664} C_VEL
LIN {X 0,Y 453.674,Z 263.598,A -85,B 0,C 180,E1 -8286.226,E2 -8286.226} C_VEL
LIN {X 0,Y 453.589,Z 263.61,A -85,B 0,C 180,E1 -8288.914,E2 -8288.914} C_VEL
LIN {X 0,Y 453.56,Z 263.613,A -85,B 0,C 180,E1 -8292.53,E2 -8292.53} C_VEL
LIN {X 0,Y 453.541,Z 263.617,A -85,B 0,C 180,E1 -8296.197,E2 -8296.197} C_VEL
LIN {X 0,Y 453.518,Z 263.619,A -85,B 0,C 180,E1 -8299.042,E2 -8299.042} C_VEL
LIN {X 0,Y 453.474,Z 263.625,A -85,B 0,C 180,E1 -8301.837,E2 -8301.837} C_VEL
LIN {X 0,Y 453.512,Z 263.621,A -85,B 0,C 180,E1 -8304.735,E2 -8304.735} C_VEL
LIN {X 0,Y 453.535,Z 263.62,A -85,B 0,C 180,E1 -8307.962,E2 -8307.962} C_VEL
LIN {X 0,Y 453.463,Z 263.631,A -85,B 0,C 180,E1 -8311.526,E2 -8311.526} C_VEL
LIN {X 0,Y 453.485,Z 263.631,A -85,B 0,C 180,E1 -8314.778,E2 -8314.778} C_VEL
LIN {X 0,Y 453.463,Z 263.631,A -85,B 0,C 180,E1 -8318.312,E2 -8318.312} C_VEL
LIN {X 0,Y 453.488,Z 263.627,A -85,B 0,C 180,E1 -8321.05,E2 -8321.05} C_VEL
LIN {X 0,Y 454.572,Z 269.709,A -85,B 0,C 180,E1 -8324.669,E2 -8324.669} C_VEL
LIN {X 0,Y 455.416,Z 274.468,A -85,B 0,C 180,E1 -8327.235,E2 -8327.235} C_VEL
LIN {X 0,Y 455.557,Z 278.219,A -85,B 0,C 180,E1 -8329.108,E2 -8329.108} C_VEL
LIN {X 0,Y 455.174,Z 284.386,A -85,B 0,C 180,E1 -8331.949,E2 -8331.949} C_VEL
LIN {X 0,Y 454.704,Z 291.691,A -85,B 0,C 180,E1 -8335.119,E2 -8335.119} C_VEL
LIN {X 0,Y 454.399,Z 298.058,A -85,B 0,C 180,E1 -8337.752,E2 -8337.752} C_VEL
LIN {X 0,Y 454.126,Z 305.786,A -85,B 0,C 180,E1 -8340.825,E2 -8340.825} C_VEL
LIN {X 0,Y 453.793,Z 314.908,A -85,B 0,C 180,E1 -8344.302,E2 -8344.302} C_VEL
LIN {X 0,Y 453.483,Z 323.672,A -85,B 0,C 180,E1 -8347.501,E2 -8347.501} C_VEL
LIN {X 0,Y 457.156,Z 338.704,A -85,B 0,C 180,E1 -8348.004,E2 -8348.004} C_VEL
LIN {X 0,Y 460.375,Z 352.804,A -85,B 0,C 180,E1 -8348.606,E2 -8348.606} C_VEL
LIN {X 0,Y 459.677,Z 367.264,A -85,B 0,C 180,E1 -8349.204,E2 -8349.204} C_VEL
LIN {X 0,Y 458.852,Z 381.298,A -85,B 0,C 180,E1 -8349.959,E2 -8349.959} C_VEL
LIN {X 0,Y 457.914,Z 394.587,A -85,B 0,C 180,E1 -8350.85,E2 -8350.85} C_VEL
LIN {X 0,Y 456.947,Z 408.139,A -85,B 0,C 180,E1 -8351.97,E2 -8351.97} C_VEL
LIN {X 0,Y 456.096,Z 420.501,A -85,B 0,C 180,E1 -8353.207,E2 -8353.207} C_VEL
LIN {X 0,Y 455.162,Z 431.789,A -85,B 0,C 180,E1 -8354.553,E2 -8354.553} C_VEL
LIN {X 0,Y 454.322,Z 442.757,A -85,B 0,C 180,E1 -8356.128,E2 -8356.128} C_VEL
LIN {X 0,Y 453.656,Z 451.899,A -85,B 0,C 180,E1 -8357.702,E2 -8357.702} C_VEL
LIN {X 0,Y 453.379,Z 458.471,A -85,B 0,C 180,E1 -8359.054,E2 -8359.054} C_VEL
LIN {X 0,Y 452.946,Z 464.937,A -85,B 0,C 180,E1 -8360.624,E2 -8360.624} C_VEL
LIN {X 0,Y 452.699,Z 470.888,A -85,B 0,C 180,E1 -8362.418,E2 -8362.418} C_VEL
LIN {X 0,Y 452.632,Z 474.387,A -85,B 0,C 180,E1 -8363.761,E2 -8363.761} C_VEL
LIN {X 0,Y 452.459,Z 477.887,A -85,B 0,C 180,E1 -8365.546,E2 -8365.546} C_VEL
LIN {X 0,Y 452.485,Z 480.189,A -85,B 0,C 180,E1 -8367.33,E2 -8367.33} C_VEL
LIN {X 0,Y 452.401,Z 481.347,A -85,B 0,C 180,E1 -8369.11,E2 -8369.11} C_VEL
LIN {X 0,Y 452.401,Z 481.346,A -85,B 0,C 180,E1 -8370.891,E2 -8370.891} C_VEL
LIN {X 0,Y 452.485,Z 480.184,A -85,B 0,C 180,E1 -8372.671,E2 -8372.671} C_VEL
LIN {X 0,Y 452.459,Z 477.88,A -85,B 0,C 180,E1 -8374.455,E2 -8374.455} C_VEL
LIN {X 0,Y 452.611,Z 474.013,A -85,B 0,C 180,E1 -8376.396,E2 -8376.396} C_VEL
LIN {X 0,Y 452.746,Z 469.547,A -85,B 0,C 180,E1 -8378.032,E2 -8378.032} C_VEL
LIN {X 0,Y 453.015,Z 463.237,A -85,B 0,C 180,E1 -8379.826,E2 -8379.826} C_VEL
LIN {X 0,Y 453.575,Z 455.33,A -85,B 0,C 180,E1 -8381.621,E2 -8381.621} C_VEL
LIN {X 0,Y 454.041,Z 447.052,A -85,B 0,C 180,E1 -8383.176,E2 -8383.176} C_VEL
LIN {X 0,Y 454.798,Z 436.8,A -85,B 0,C 180,E1 -8384.773,E2 -8384.773} C_VEL
LIN {X 0,Y 455.547,Z 426.462,A -85,B 0,C 180,E1 -8386.123,E2 -8386.123} C_VEL
LIN {X 0,Y 456.55,Z 414.133,A -85,B 0,C 180,E1 -8387.472,E2 -8387.472} C_VEL
LIN {X 0,Y 457.517,Z 400.474,A -85,B 0,C 180,E1 -8388.704,E2 -8388.704} C_VEL
LIN {X 0,Y 458.453,Z 386.774,A -85,B 0,C 180,E1 -8389.71,E2 -8389.71} C_VEL
LIN {X 0,Y 459.395,Z 372.61,A -85,B 0,C 180,E1 -8390.543,E2 -8390.543} C_VEL
LIN {X 0,Y 460.173,Z 357.195,A -85,B 0,C 180,E1 -8391.244,E2 -8391.244} C_VEL
LIN {X 0,Y 460.234,Z 351.958,A -85,B 0,C 180,E1 -8391.442,E2 -8391.442} C_VEL
LIN {X 0,Y 456.692,Z 336.915,A -85,B 0,C 180,E1 -8392.072,E2 -8392.072} C_VEL
LIN {X 0,Y 453.499,Z 323.933,A -85,B 0,C 180,E1 -8392.5,E2 -8392.5} C_VEL
LIN {X 0,Y 453.826,Z 315.499,A -85,B 0,C 180,E1 -8395.698,E2 -8395.698} C_VEL
LIN {X 0,Y 454.145,Z 307.771,A -85,B 0,C 180,E1 -8398.669,E2 -8398.669} C_VEL
LIN {X 0,Y 454.439,Z 300.088,A -85,B 0,C 180,E1 -8401.724,E2 -8401.724} C_VEL
LIN {X 0,Y 454.819,Z 292.492,A -85,B 0,C 180,E1 -8404.872,E2 -8404.872} C_VEL
LIN {X 0,Y 455.297,Z 285.113,A -85,B 0,C 180,E1 -8408.071,E2 -8408.071} C_VEL
LIN {X 0,Y 455.626,Z 278.878,A -85,B 0,C 180,E1 -8410.902,E2 -8410.902} C_VEL
LIN {X 0,Y 455.475,Z 275.026,A -85,B 0,C 180,E1 -8412.76,E2 -8412.76} C_VEL
LIN {X 0,Y 454.477,Z 269.002,A -85,B 0,C 180,E1 -8415.902,E2 -8415.902} C_VEL
LIN {X 0,Y 453.503,Z 263.623,A -85,B 0,C 180,E1 -8418.951,E2 -8418.951} C_VEL
LIN {X 0,Y 453.47,Z 263.627,A -85,B 0,C 180,E1 -8421.688,E2 -8421.688} C_VEL
LIN {X 0,Y 453.488,Z 263.624,A -85,B 0,C 180,E1 -8425.224,E2 -8425.224} C_VEL
LIN {X 0,Y 453.471,Z 263.625,A -85,B 0,C 180,E1 -8428.475,E2 -8428.475} C_VEL
LIN {X 0,Y 453.537,Z 263.615,A -85,B 0,C 180,E1 -8432.04,E2 -8432.04} C_VEL
LIN {X 0,Y 453.519,Z 263.618,A -85,B 0,C 180,E1 -8435.265,E2 -8435.265} C_VEL
LIN {X 0,Y 453.486,Z 263.624,A -85,B 0,C 180,E1 -8438.415,E2 -8438.415} C_VEL
LIN {X 0,Y 453.528,Z 263.619,A -85,B 0,C 180,E1 -8441.008,E2 -8441.008} C_VEL
LIN {X 0,Y 453.575,Z 263.611,A -85,B 0,C 180,E1 -8443.879,E2 -8443.879} C_VEL
LIN {X 0,Y 453.569,Z 263.611,A -85,B 0,C 180,E1 -8447.471,E2 -8447.471} C_VEL
LIN {X 0,Y 453.596,Z 263.609,A -85,B 0,C 180,E1 -8451.086,E2 -8451.086} C_VEL
LIN {X 0,Y 453.656,Z 263.6,A -85,B 0,C 180,E1 -8453.774,E2 -8453.774} C_VEL
LIN {X 0,Y 453.749,Z 263.588,A -85,B 0,C 180,E1 -8457.336,E2 -8457.336} C_VEL
LIN {X 0,Y 453.828,Z 263.58,A -85,B 0,C 180,E1 -8459.999,E2 -8459.999} C_VEL
LIN {X 0,Y 453.747,Z 263.591,A -85,B 0,C 180,E1 -8462.662,E2 -8462.662} C_VEL
LIN {X 0,Y 453.68,Z 263.6,A -85,B 0,C 180,E1 -8466.224,E2 -8466.224} C_VEL
LIN {X 0,Y 453.595,Z 263.608,A -85,B 0,C 180,E1 -8468.912,E2 -8468.912} C_VEL
LIN {X 0,Y 453.566,Z 263.615,A -85,B 0,C 180,E1 -8472.528,E2 -8472.528} C_VEL
LIN {X 0,Y 453.547,Z 263.617,A -85,B 0,C 180,E1 -8476.195,E2 -8476.195} C_VEL
LIN {X 0,Y 453.521,Z 263.617,A -85,B 0,C 180,E1 -8479.039,E2 -8479.039} C_VEL
LIN {X 0,Y 453.477,Z 263.625,A -85,B 0,C 180,E1 -8481.835,E2 -8481.835} C_VEL
LIN {X 0,Y 453.514,Z 263.619,A -85,B 0,C 180,E1 -8484.733,E2 -8484.733} C_VEL
LIN {X 0,Y 453.537,Z 263.618,A -85,B 0,C 180,E1 -8487.96,E2 -8487.96} C_VEL
LIN {X 0,Y 453.464,Z 263.625,A -85,B 0,C 180,E1 -8491.524,E2 -8491.524} C_VEL
LIN {X 0,Y 453.487,Z 263.621,A -85,B 0,C 180,E1 -8494.776,E2 -8494.776} C_VEL
LIN {X 0,Y 453.47,Z 263.626,A -85,B 0,C 180,E1 -8498.309,E2 -8498.309} C_VEL
LIN {X 0,Y 453.49,Z 263.621,A -85,B 0,C 180,E1 -8500.607,E2 -8500.607} C_VEL
LIN {X 0,Y 453.458,Z 263.626,A -85,B 0,C 180,E1 -8503.244,E2 -8503.244} C_VEL
LIN {X 0,Y 453.472,Z 263.626,A -85,B 0,C 180,E1 -8505.779,E2 -8505.779} C_VEL
LIN {X 0,Y 453.491,Z 263.622,A -85,B 0,C 180,E1 -8508.21,E2 -8508.21} C_VEL
LIN {X 0,Y 453.52,Z 263.616,A -85,B 0,C 180,E1 -8510.787,E2 -8510.787} C_VEL
LIN {X 0,Y 453.451,Z 263.628,A -85,B 0,C 180,E1 -8513.916,E2 -8513.916} C_VEL
LIN {X 0,Y 453.476,Z 263.624,A -85,B 0,C 180,E1 -8517.15,E2 -8517.15} C_VEL
LIN {X 0,Y 453.506,Z 263.62,A -85,B 0,C 180,E1 -8520.27,E2 -8520.27} C_VEL
LIN {X 0,Y 453.506,Z 263.622,A -85,B 0,C 180,E1 -8523.293,E2 -8523.293} C_VEL
LIN {X 0,Y 453.495,Z 263.62,A -85,B 0,C 180,E1 -8526.238,E2 -8526.238} C_VEL
LIN {X 0,Y 453.474,Z 263.625,A -85,B 0,C 180,E1 -8529.117,E2 -8529.117} C_VEL
LIN {X 0,Y 453.502,Z 263.622,A -85,B 0,C 180,E1 -8531.944,E2 -8531.944} C_VEL
LIN {X 0,Y 453.531,Z 263.616,A -85,B 0,C 180,E1 -8534.725,E2 -8534.725} C_VEL
LIN {X 0,Y 453.592,Z 263.612,A -85,B 0,C 180,E1 -8537.471,E2 -8537.471} C_VEL
LIN {X 0,Y 453.584,Z 263.612,A -85,B 0,C 180,E1 -8541.086,E2 -8541.086} C_VEL
LIN {X 0,Y 453.624,Z 263.605,A -85,B 0,C 180,E1 -8543.085,E2 -8543.085} C_VEL
LIN {X 0,Y 452.93,Z 263.693,A -85,B 0,C 180,E1 -8543.825,E2 -8543.825} C_VEL
LIN {X 0,Y 449.926,Z 264.068,A -85,B 0,C 180,E1 -8545.025,E2 -8545.025} C_VEL
LIN {X 0,Y 447.365,Z 264.385,A -85,B 0,C 180,E1 -8545.992,E2 -8545.992} C_VEL
LIN {X 0,Y 446.247,Z 264.526,A -85,B 0,C 180,E1 -8546.742,E2 -8546.742} C_VEL
LIN {X 0,Y 446.146,Z 264.538,A -85,B 0,C 180,E1 -8546.997,E2 -8546.997} C_VEL
LIN {X 0,Y 446.273,Z 264.524,A -85,B 0,C 180,E1 -8548.194,E2 -8548.194} C_VEL
LIN {X 0,Y 446.459,Z 264.88,A -85,B 0,C 180,E1 -8549.097,E2 -8549.097} C_VEL
LIN {X 0,Y 445.953,Z 268.97,A -85,B 0,C 180,E1 -8553.614,E2 -8553.614} C_VEL
LIN {X 0,Y 445.913,Z 271.443,A -85,B 0,C 180,E1 -8556.333,E2 -8556.333} C_VEL
LIN {X 0,Y 445.813,Z 273.954,A -85,B 0,C 180,E1 -8559.07,E2 -8559.07} C_VEL
LIN {X 0,Y 445.786,Z 275.053,A -85,B 0,C 180,E1 -8560.244,E2 -8560.244} C_VEL
LIN {X 0,Y 447.548,Z 280.375,A -85,B 0,C 180,E1 -8560.461,E2 -8560.461} C_VEL
LIN {X 0,Y 451.983,Z 293.929,A -85,B 0,C 180,E1 -8561.077,E2 -8561.077} C_VEL
LIN {X 0,Y 453.896,Z 300.72,A -85,B 0,C 180,E1 -8561.425,E2 -8561.425} C_VEL
LIN {X 0,Y 453.175,Z 315.504,A -85,B 0,C 180,E1 -8562.07,E2 -8562.07} C_VEL
LIN {X 0,Y 452.337,Z 330.076,A -85,B 0,C 180,E1 -8562.905,E2 -8562.905} C_VEL
LIN {X 0,Y 451.446,Z 343.231,A -85,B 0,C 180,E1 -8563.848,E2 -8563.848} C_VEL
LIN {X 0,Y 450.56,Z 356.115,A -85,B 0,C 180,E1 -8564.979,E2 -8564.979} C_VEL
LIN {X 0,Y 449.598,Z 367.917,A -85,B 0,C 180,E1 -8566.225,E2 -8566.225} C_VEL
LIN {X 0,Y 448.73,Z 378.435,A -85,B 0,C 180,E1 -8567.547,E2 -8567.547} C_VEL
LIN {X 0,Y 447.887,Z 388.194,A -85,B 0,C 180,E1 -8569.001,E2 -8569.001} C_VEL
LIN {X 0,Y 447.148,Z 397.669,A -85,B 0,C 180,E1 -8570.709,E2 -8570.709} C_VEL
LIN {X 0,Y 446.608,Z 404.506,A -85,B 0,C 180,E1 -8572.189,E2 -8572.189} C_VEL
LIN {X 0,Y 446.134,Z 411.323,A -85,B 0,C 180,E1 -8573.985,E2 -8573.985} C_VEL
LIN {X 0,Y 445.848,Z 416.234,A -85,B 0,C 180,E1 -8575.609,E2 -8575.609} C_VEL
LIN {X 0,Y 445.68,Z 420.067,A -85,B 0,C 180,E1 -8577.213,E2 -8577.213} C_VEL
LIN {X 0,Y 445.427,Z 423.566,A -85,B 0,C 180,E1 -8579.282,E2 -8579.282} C_VEL
LIN {X 0,Y 445.373,Z 424.75,A -85,B 0,C 180,E1 -8580.328,E2 -8580.328} C_VEL
LIN {X 0,Y 445.336,Z 425.652,A -85,B 0,C 180,E1 -8581.552,E2 -8581.552} C_VEL
LIN {X 0,Y 445.315,Z 426.031,A -85,B 0,C 180,E1 -8583.529,E2 -8583.529} C_VEL
LIN {X 0,Y 445.342,Z 425.549,A -85,B 0,C 180,E1 -8584.856,E2 -8584.856} C_VEL
LIN {X 0,Y 445.414,Z 423.673,A -85,B 0,C 180,E1 -8586.839,E2 -8586.839} C_VEL
LIN {X 0,Y 445.64,Z 420.953,A -85,B 0,C 180,E1 -8588.53,E2 -8588.53} C_VEL
LIN {X 0,Y 445.846,Z 417.095,A -85,B 0,C 180,E1 -8590.262,E2 -8590.262} C_VEL
LIN {X 0,Y 446.209,Z 411.177,A -85,B 0,C 180,E1 -8592.248,E2 -8592.248} C_VEL
LIN {X 0,Y 446.683,Z 404.037,A -85,B 0,C 180,E1 -8594.112,E2 -8594.112} C_VEL
LIN {X 0,Y 447.304,Z 396.905,A -85,B 0,C 180,E1 -8595.633,E2 -8595.633} C_VEL
LIN {X 0,Y 448.003,Z 388.307,A -85,B 0,C 180,E1 -8597.17,E2 -8597.17} C_VEL
LIN {X 0,Y 448.894,Z 377.869,A -85,B 0,C 180,E1 -8598.719,E2 -8598.719} C_VEL
LIN {X 0,Y 449.925,Z 365.97,A -85,B 0,C 180,E1 -8600.178,E2 -8600.178} C_VEL
LIN {X 0,Y 450.972,Z 353.518,A -85,B 0,C 180,E1 -8601.44,E2 -8601.44} C_VEL
LIN {X 0,Y 451.935,Z 339.642,A -85,B 0,C 180,E1 -8602.594,E2 -8602.594} C_VEL
LIN {X 0,Y 452.897,Z 326.024,A -85,B 0,C 180,E1 -8603.503,E2 -8603.503} C_VEL
LIN {X 0,Y 453.635,Z 311.379,A -85,B 0,C 180,E1 -8604.278,E2 -8604.278} C_VEL
LIN {X 0,Y 454.003,Z 300.802,A -85,B 0,C 180,E1 -8604.72,E2 -8604.72} C_VEL
LIN {X 0,Y 449.437,Z 286.474,A -85,B 0,C 180,E1 -8605.438,E2 -8605.438} C_VEL
LIN {X 0,Y 445.996,Z 277.002,A -85,B 0,C 180,E1 -8605.851,E2 -8605.851} C_VEL
LIN {X 0,Y 445.879,Z 276.362,A -85,B 0,C 180,E1 -8605.909,E2 -8605.909} C_VEL
LIN {X 0,Y 445.958,Z 273.982,A -85,B 0,C 180,E1 -8608.665,E2 -8608.665} C_VEL
LIN {X 0,Y 446.039,Z 271.203,A -85,B 0,C 180,E1 -8611.927,E2 -8611.927} C_VEL
LIN {X 0,Y 446.143,Z 268.763,A -85,B 0,C 180,E1 -8614.83,E2 -8614.83} C_VEL
LIN {X 0,Y 446.209,Z 265.832,A -85,B 0,C 180,E1 -8618.32,E2 -8618.32} C_VEL
LIN {X 0,Y 446.227,Z 264.682,A -85,B 0,C 180,E1 -8619.728,E2 -8619.728} C_VEL
LIN {X 0,Y 446.381,Z 264.512,A -85,B 0,C 180,E1 -8621.647,E2 -8621.647} C_VEL
LIN {X 0,Y 446.5,Z 264.497,A -85,B 0,C 180,E1 -8624.481,E2 -8624.481} C_VEL
LIN {X 0,Y 446.511,Z 264.492,A -85,B 0,C 180,E1 -8628.194,E2 -8628.194} C_VEL
LIN {X 0,Y 446.594,Z 264.484,A -85,B 0,C 180,E1 -8631.859,E2 -8631.859} C_VEL
LIN {X 0,Y 446.642,Z 264.476,A -85,B 0,C 180,E1 -8634.584,E2 -8634.584} C_VEL
LIN {X 0,Y 446.705,Z 264.468,A -85,B 0,C 180,E1 -8637.296,E2 -8637.296} C_VEL
LIN {X 0,Y 446.789,Z 264.456,A -85,B 0,C 180,E1 -8640.001,E2 -8640.001} C_VEL
LIN {X 0,Y 446.705,Z 264.469,A -85,B 0,C 180,E1 -8642.706,E2 -8642.706} C_VEL
LIN {X 0,Y 446.643,Z 264.474,A -85,B 0,C 180,E1 -8646.325,E2 -8646.325} C_VEL
LIN {X 0,Y 446.535,Z 264.49,A -85,B 0,C 180,E1 -8649.056,E2 -8649.056} C_VEL
LIN {X 0,Y 446.518,Z 264.49,A -85,B 0,C 180,E1 -8652.731,E2 -8652.731} C_VEL
LIN {X 0,Y 446.493,Z 264.495,A -85,B 0,C 180,E1 -8656.229,E2 -8656.229} C_VEL
LIN {X 0,Y 446.467,Z 264.496,A -85,B 0,C 180,E1 -8659.304,E2 -8659.304} C_VEL
LIN {X 0,Y 446.416,Z 264.504,A -85,B 0,C 180,E1 -8662.2,E2 -8662.2} C_VEL
LIN {X 0,Y 446.456,Z 264.498,A -85,B 0,C 180,E1 -8665.153,E2 -8665.153} C_VEL
LIN {X 0,Y 446.482,Z 264.498,A -85,B 0,C 180,E1 -8668.18,E2 -8668.18} C_VEL
LIN {X 0,Y 446.417,Z 264.51,A -85,B 0,C 180,E1 -8671.776,E2 -8671.776} C_VEL
LIN {X 0,Y 446.427,Z 264.51,A -85,B 0,C 180,E1 -8674.524,E2 -8674.524} C_VEL
LIN {X 0,Y 446.414,Z 264.509,A -85,B 0,C 180,E1 -8678.08,E2 -8678.08} C_VEL
LIN {X 0,Y 446.468,Z 264.681,A -85,B 0,C 180,E1 -8680.706,E2 -8680.706} C_VEL
LIN {X 0,Y 447.314,Z 269.596,A -85,B 0,C 180,E1 -8683.734,E2 -8683.734} C_VEL
LIN {X 0,Y 448.219,Z 274.235,A -85,B 0,C 180,E1 -8686.378,E2 -8686.378} C_VEL
LIN {X 0,Y 448.595,Z 278.836,A -85,B 0,C 180,E1 -8688.765,E2 -8688.765} C_VEL
LIN {X 0,Y 448.226,Z 284.898,A -85,B 0,C 180,E1 -8691.627,E2 -8691.627} C_VEL
LIN {X 0,Y 447.715,Z 291.857,A -85,B 0,C 180,E1 -8694.714,E2 -8694.714} C_VEL
LIN {X 0,Y 447.389,Z 298.99,A -85,B 0,C 180,E1 -8697.718,E2 -8697.718} C_VEL
LIN {X 0,Y 447.075,Z 306.661,A -85,B 0,C 180,E1 -8700.836,E2 -8700.836} C_VEL
LIN {X 0,Y 446.71,Z 315.714,A -85,B 0,C 180,E1 -8704.365,E2 -8704.365} C_VEL
LIN {X 0,Y 446.411,Z 323.02,A -85,B 0,C 180,E1 -8707.12,E2 -8707.12} C_VEL
LIN {X 0,Y 450.306,Z 339.306,A -85,B 0,C 180,E1 -8707.681,E2 -8707.681} C_VEL
LIN {X 0,Y 453.607,Z 353.629,A -85,B 0,C 180,E1 -8708.323,E2 -8708.323} C_VEL
LIN {X 0,Y 452.874,Z 369.004,A -85,B 0,C 180,E1 -8708.995,E2 -8708.995} C_VEL
LIN {X 0,Y 452.001,Z 382.573,A -85,B 0,C 180,E1 -8709.76,E2 -8709.76} C_VEL
LIN {X 0,Y 450.914,Z 396.96,A -85,B 0,C 180,E1 -8710.777,E2 -8710.777} C_VEL
LIN {X 0,Y 449.907,Z 410.007,A -85,B 0,C 180,E1 -8711.913,E2 -8711.913} C_VEL
LIN {X 0,Y 449.039,Z 421.982,A -85,B 0,C 180,E1 -8713.17,E2 -8713.17} C_VEL
LIN {X 0,Y 448.068,Z 432.953,A -85,B 0,C 180,E1 -8714.536,E2 -8714.536} C_VEL
LIN {X 0,Y 447.224,Z 443.65,A -85,B 0,C 180,E1 -8716.135,E2 -8716.135} C_VEL
LIN {X 0,Y 446.564,Z 452.615,A -85,B 0,C 180,E1 -8717.745,E2 -8717.745} C_VEL
LIN {X 0,Y 446.25,Z 459.026,A -85,B 0,C 180,E1 -8719.107,E2 -8719.107} C_VEL
LIN {X 0,Y 445.802,Z 466.117,A -85,B 0,C 180,E1 -8720.93,E2 -8720.93} C_VEL
LIN {X 0,Y 445.587,Z 471.701,A -85,B 0,C 180,E1 -8722.752,E2 -8722.752} C_VEL
LIN {X 0,Y 445.475,Z 475.926,A -85,B 0,C 180,E1 -8724.569,E2 -8724.569} C_VEL
LIN {X 0,Y 445.34,Z 478.884,A -85,B 0,C 180,E1 -8726.381,E2 -8726.381} C_VEL
LIN {X 0,Y 445.349,Z 480.654,A -85,B 0,C 180,E1 -8728.192,E2 -8728.192} C_VEL
LIN {X 0,Y 445.29,Z 481.257,A -85,B 0,C 180,E1 -8730.001,E2 -8730.001} C_VEL
LIN {X 0,Y 445.35,Z 480.654,A -85,B 0,C 180,E1 -8731.809,E2 -8731.809} C_VEL
LIN {X 0,Y 445.34,Z 478.884,A -85,B 0,C 180,E1 -8733.62,E2 -8733.62} C_VEL
LIN {X 0,Y 445.465,Z 475.934,A -85,B 0,C 180,E1 -8735.432,E2 -8735.432} C_VEL
LIN {X 0,Y 445.587,Z 471.723,A -85,B 0,C 180,E1 -8737.249,E2 -8737.249} C_VEL
LIN {X 0,Y 445.803,Z 466.148,A -85,B 0,C 180,E1 -8739.071,E2 -8739.071} C_VEL
LIN {X 0,Y 446.248,Z 459.065,A -85,B 0,C 180,E1 -8740.894,E2 -8740.894} C_VEL
LIN {X 0,Y 446.675,Z 451.126,A -85,B 0,C 180,E1 -8742.564,E2 -8742.564} C_VEL
LIN {X 0,Y 447.356,Z 442.367,A -85,B 0,C 180,E1 -8744.094,E2 -8744.094} C_VEL
LIN {X 0,Y 448.225,Z 431.417,A -85,B 0,C 180,E1 -8745.693,E2 -8745.693} C_VEL
LIN {X 0,Y 449.23,Z 419.12,A -85,B 0,C 180,E1 -8747.176,E2 -8747.176} C_VEL
LIN {X 0,Y 450.23,Z 406.595,A -85,B 0,C 180,E1 -8748.428,E2 -8748.428} C_VEL
LIN {X 0,Y 451.267,Z 392.755,A -85,B 0,C 180,E1 -8749.563,E2 -8749.563} C_VEL
LIN {X 0,Y 452.254,Z 379.188,A -85,B 0,C 180,E1 -8750.466,E2 -8750.466} C_VEL
LIN {X 0,Y 453.152,Z 364.764,A -85,B 0,C 180,E1 -8751.228,E2 -8751.228} C_VEL
LIN {X 0,Y 453.531,Z 353.301,A -85,B 0,C 180,E1 -8751.705,E2 -8751.705} C_VEL
LIN {X 0,Y 450.031,Z 338.193,A -85,B 0,C 180,E1 -8752.372,E2 -8752.372} C_VEL
LIN {X 0,Y 446.453,Z 323.497,A -85,B 0,C 180,E1 -8752.879,E2 -8752.879} C_VEL
LIN {X 0,Y 446.782,Z 315.061,A -85,B 0,C 180,E1 -8756.133,E2 -8756.133} C_VEL
LIN {X 0,Y 447.134,Z 307.355,A -85,B 0,C 180,E1 -8759.161,E2 -8759.161} C_VEL
LIN {X 0,Y 447.461,Z 299.76,A -85,B 0,C 180,E1 -8762.278,E2 -8762.278} C_VEL
LIN {X 0,Y 447.864,Z 292.613,A -85,B 0,C 180,E1 -8765.313,E2 -8765.313} C_VEL
LIN {X 0,Y 448.332,Z 285.64,A -85,B 0,C 180,E1 -8768.39,E2 -8768.39} C_VEL
LIN {X 0,Y 448.684,Z 279.516,A -85,B 0,C 180,E1 -8771.248,E2 -8771.248} C_VEL
LIN {X 0,Y 448.436,Z 275.89,A -85,B 0,C 180,E1 -8773.043,E2 -8773.043} C_VEL
LIN {X 0,Y 447.62,Z 270.91,A -85,B 0,C 180,E1 -8775.678,E2 -8775.678} C_VEL
LIN {X 0,Y 446.684,Z 265.663,A -85,B 0,C 180,E1 -8778.637,E2 -8778.637} C_VEL
LIN {X 0,Y 446.466,Z 264.499,A -85,B 0,C 180,E1 -8779.436,E2 -8779.436} C_VEL
LIN {X 0,Y 446.414,Z 264.504,A -85,B 0,C 180,E1 -8782.121,E2 -8782.121} C_VEL
LIN {X 0,Y 446.428,Z 264.504,A -85,B 0,C 180,E1 -8785.476,E2 -8785.476} C_VEL
LIN {X 0,Y 446.421,Z 264.505,A -85,B 0,C 180,E1 -8788.699,E2 -8788.699} C_VEL
LIN {X 0,Y 446.491,Z 264.492,A -85,B 0,C 180,E1 -8791.821,E2 -8791.821} C_VEL
LIN {X 0,Y 446.464,Z 264.5,A -85,B 0,C 180,E1 -8794.847,E2 -8794.847} C_VEL
LIN {X 0,Y 446.454,Z 264.498,A -85,B 0,C 180,E1 -8798.245,E2 -8798.245} C_VEL
LIN {X 0,Y 446.463,Z 264.496,A -85,B 0,C 180,E1 -8801.649,E2 -8801.649} C_VEL
LIN {X 0,Y 446.513,Z 264.493,A -85,B 0,C 180,E1 -8804.479,E2 -8804.479} C_VEL
LIN {X 0,Y 446.522,Z 264.491,A -85,B 0,C 180,E1 -8808.192,E2 -8808.192} C_VEL
LIN {X 0,Y 446.542,Z 264.488,A -85,B 0,C 180,E1 -8810.944,E2 -8810.944} C_VEL
LIN {X 0,Y 446.624,Z 264.475,A -85,B 0,C 180,E1 -8813.675,E2 -8813.675} C_VEL
LIN {X 0,Y 446.696,Z 264.466,A -85,B 0,C 180,E1 -8817.294,E2 -8817.294} C_VEL
LIN {X 0,Y 446.798,Z 264.456,A -85,B 0,C 180,E1 -8819.999,E2 -8819.999} C_VEL
LIN {X 0,Y 446.694,Z 264.47,A -85,B 0,C 180,E1 -8822.704,E2 -8822.704} C_VEL
LIN {X 0,Y 446.65,Z 264.477,A -85,B 0,C 180,E1 -8826.323,E2 -8826.323} C_VEL
LIN {X 0,Y 446.541,Z 264.486,A -85,B 0,C 180,E1 -8829.054,E2 -8829.054} C_VEL
LIN {X 0,Y 446.524,Z 264.49,A -85,B 0,C 180,E1 -8832.728,E2 -8832.728} C_VEL
LIN {X 0,Y 446.498,Z 264.495,A -85,B 0,C 180,E1 -8836.227,E2 -8836.227} C_VEL
LIN {X 0,Y 446.47,Z 264.495,A -85,B 0,C 180,E1 -8839.302,E2 -8839.302} C_VEL
LIN {X 0,Y 446.419,Z 264.505,A -85,B 0,C 180,E1 -8842.198,E2 -8842.198} C_VEL
LIN {X 0,Y 446.457,Z 264.496,A -85,B 0,C 180,E1 -8845.151,E2 -8845.151} C_VEL
LIN {X 0,Y 446.484,Z 264.497,A -85,B 0,C 180,E1 -8848.177,E2 -8848.177} C_VEL
LIN {X 0,Y 446.417,Z 264.505,A -85,B 0,C 180,E1 -8851.774,E2 -8851.774} C_VEL
LIN {X 0,Y 446.428,Z 264.502,A -85,B 0,C 180,E1 -8854.521,E2 -8854.521} C_VEL
LIN {X 0,Y 446.427,Z 264.503,A -85,B 0,C 180,E1 -8858.08,E2 -8858.08} C_VEL
LIN {X 0,Y 446.424,Z 264.501,A -85,B 0,C 180,E1 -8860.916,E2 -8860.916} C_VEL
LIN {X 0,Y 446.418,Z 264.505,A -85,B 0,C 180,E1 -8863.842,E2 -8863.842} C_VEL
LIN {X 0,Y 446.442,Z 264.499,A -85,B 0,C 180,E1 -8866.396,E2 -8866.396} C_VEL
LIN {X 0,Y 446.462,Z 264.499,A -85,B 0,C 180,E1 -8869.803,E2 -8869.803} C_VEL
LIN {X 0,Y 446.426,Z 264.503,A -85,B 0,C 180,E1 -8872.122,E2 -8872.122} C_VEL
LIN {X 0,Y 446.424,Z 264.504,A -85,B 0,C 180,E1 -8875.476,E2 -8875.476} C_VEL
LIN {X 0,Y 446.412,Z 264.502,A -85,B 0,C 180,E1 -8878.699,E2 -8878.699} C_VEL
LIN {X 0,Y 446.476,Z 264.498,A -85,B 0,C 180,E1 -8881.82,E2 -8881.82} C_VEL
LIN {X 0,Y 446.449,Z 264.497,A -85,B 0,C 180,E1 -8884.847,E2 -8884.847} C_VEL
LIN {X 0,Y 446.439,Z 264.499,A -85,B 0,C 180,E1 -8888.244,E2 -8888.244} C_VEL
LIN {X 0,Y 446.448,Z 264.501,A -85,B 0,C 180,E1 -8891.648,E2 -8891.648} C_VEL
LIN {X 0,Y 446.498,Z 264.491,A -85,B 0,C 180,E1 -8894.479,E2 -8894.479} C_VEL
LIN {X 0,Y 446.53,Z 264.488,A -85,B 0,C 180,E1 -8898.193,E2 -8898.193} C_VEL
LIN {X 0,Y 446.59,Z 264.481,A -85,B 0,C 180,E1 -8901.857,E2 -8901.857} C_VEL
LIN {X 0,Y 446.62,Z 264.476,A -85,B 0,C 180,E1 -8904.582,E2 -8904.582} C_VEL
LIN {X 0,Y 446.146,Z 264.538,A -85,B 0,C 180,E1 -8906.997,E2 -8906.997} C_VEL
LIN {X 0,Y 445.484,Z 264.706,A -85,B 0,C 180,E1 -8907.751,E2 -8907.751} C_VEL
LIN {X 0,Y 442.718,Z 265.506,A -85,B 0,C 180,E1 -8908.975,E2 -8908.975} C_VEL
LIN {X 0,Y 440.315,Z 266.422,A -85,B 0,C 180,E1 -8909.96,E2 -8909.96} C_VEL
LIN {X 0,Y 439.18,Z 267.157,A -85,B 0,C 180,E1 -8910.718,E2 -8910.718} C_VEL
LIN {X 0,Y 439.031,Z 267.396,A -85,B 0,C 180,E1 -8910.976,E2 -8910.976} C_VEL
LIN {X 0,Y 438.942,Z 270.629,A -85,B 0,C 180,E1 -8914.591,E2 -8914.591} C_VEL
LIN {X 0,Y 438.862,Z 273.141,A -85,B 0,C 180,E1 -8917.36,E2 -8917.36} C_VEL
LIN {X 0,Y 438.738,Z 275.452,A -85,B 0,C 180,E1 -8919.857,E2 -8919.857} C_VEL
LIN {X 0,Y 441.35,Z 283.157,A -85,B 0,C 180,E1 -8920.189,E2 -8920.189} C_VEL
LIN {X 0,Y 445.602,Z 296.356,A -85,B 0,C 180,E1 -8920.823,E2 -8920.823} C_VEL
LIN {X 0,Y 447.271,Z 302.314,A -85,B 0,C 180,E1 -8921.144,E2 -8921.144} C_VEL
LIN {X 0,Y 446.482,Z 317.008,A -85,B 0,C 180,E1 -8921.807,E2 -8921.807} C_VEL
LIN {X 0,Y 445.601,Z 331.724,A -85,B 0,C 180,E1 -8922.68,E2 -8922.68} C_VEL
LIN {X 0,Y 444.63,Z 345.593,A -85,B 0,C 180,E1 -8923.715,E2 -8923.715} C_VEL
LIN {X 0,Y 443.604,Z 358.515,A -85,B 0,C 180,E1 -8924.897,E2 -8924.897} C_VEL
LIN {X 0,Y 442.589,Z 370.731,A -85,B 0,C 180,E1 -8926.252,E2 -8926.252} C_VEL
LIN {X 0,Y 441.671,Z 380.885,A -85,B 0,C 180,E1 -8927.597,E2 -8927.597} C_VEL
LIN {X 0,Y 440.823,Z 390.31,A -85,B 0,C 180,E1 -8929.076,E2 -8929.076} C_VEL
LIN {X 0,Y 440.08,Z 399.5,A -85,B 0,C 180,E1 -8930.813,E2 -8930.813} C_VEL
LIN {X 0,Y 439.503,Z 407.104,A -85,B 0,C 180,E1 -8932.567,E2 -8932.567} C_VEL
LIN {X 0,Y 439.016,Z 412.767,A -85,B 0,C 180,E1 -8934.153,E2 -8934.153} C_VEL
LIN {X 0,Y 438.785,Z 417.006,A -85,B 0,C 180,E1 -8935.623,E2 -8935.623} C_VEL
LIN {X 0,Y 438.624,Z 420.589,A -85,B 0,C 180,E1 -8937.17,E2 -8937.17} C_VEL
LIN {X 0,Y 438.395,Z 423.344,A -85,B 0,C 180,E1 -8938.746,E2 -8938.746} C_VEL
LIN {X 0,Y 438.304,Z 424.955,A -85,B 0,C 180,E1 -8940.022,E2 -8940.022} C_VEL
LIN {X 0,Y 438.246,Z 426.316,A -85,B 0,C 180,E1 -8941.951,E2 -8941.951} C_VEL
LIN {X 0,Y 438.24,Z 426.478,A -85,B 0,C 180,E1 -8943.5,E2 -8943.5} C_VEL
LIN {X 0,Y 438.268,Z 425.758,A -85,B 0,C 180,E1 -8945.259,E2 -8945.259} C_VEL
LIN {X 0,Y 438.338,Z 424.343,A -85,B 0,C 180,E1 -8946.713,E2 -8946.713} C_VEL
LIN {X 0,Y 438.6,Z 421.297,A -85,B 0,C 180,E1 -8948.676,E2 -8948.676} C_VEL
LIN {X 0,Y 438.803,Z 417.391,A -85,B 0,C 180,E1 -8950.44,E2 -8950.44} C_VEL
LIN {X 0,Y 439.15,Z 412.195,A -85,B 0,C 180,E1 -8952.232,E2 -8952.232} C_VEL
LIN {X 0,Y 439.631,Z 405.735,A -85,B 0,C 180,E1 -8953.999,E2 -8953.999} C_VEL
LIN {X 0,Y 440.274,Z 398.699,A -85,B 0,C 180,E1 -8955.565,E2 -8955.565} C_VEL
LIN {X 0,Y 440.974,Z 390.206,A -85,B 0,C 180,E1 -8957.148,E2 -8957.148} C_VEL
LIN {X 0,Y 441.871,Z 380.085,A -85,B 0,C 180,E1 -8958.721,E2 -8958.721} C_VEL
LIN {X 0,Y 442.916,Z 369.109,A -85,B 0,C 180,E1 -8960.137,E2 -8960.137} C_VEL
LIN {X 0,Y 443.958,Z 357.314,A -85,B 0,C 180,E1 -8961.408,E2 -8961.408} C_VEL
LIN {X 0,Y 444.988,Z 344.51,A -85,B 0,C 180,E1 -8962.553,E2 -8962.553} C_VEL
LIN {X 0,Y 445.894,Z 331.635,A -85,B 0,C 180,E1 -8963.497,E2 -8963.497} C_VEL
LIN {X 0,Y 446.789,Z 317.245,A -85,B 0,C 180,E1 -8964.34,E2 -8964.34} C_VEL
LIN {X 0,Y 447.387,Z 302.363,A -85,B 0,C 180,E1 -8965.015,E2 -8965.015} C_VEL
LIN {X 0,Y 442.916,Z 288.349,A -85,B 0,C 180,E1 -8965.752,E2 -8965.752} C_VEL
LIN {X 0,Y 438.954,Z 277.494,A -85,B 0,C 180,E1 -8966.245,E2 -8966.245} C_VEL
LIN {X 0,Y 438.839,Z 276.881,A -85,B 0,C 180,E1 -8966.284,E2 -8966.284} C_VEL
LIN {X 0,Y 438.898,Z 274.409,A -85,B 0,C 180,E1 -8969.177,E2 -8969.177} C_VEL
LIN {X 0,Y 438.994,Z 271.736,A -85,B 0,C 180,E1 -8972.338,E2 -8972.338} C_VEL
LIN {X 0,Y 439.123,Z 268.848,A -85,B 0,C 180,E1 -8975.818,E2 -8975.818} C_VEL
LIN {X 0,Y 439.189,Z 266.723,A -85,B 0,C 180,E1 -8978.406,E2 -8978.406} C_VEL
LIN {X 0,Y 439.247,Z 265.399,A -85,B 0,C 180,E1 -8980.368,E2 -8980.368} C_VEL
LIN {X 0,Y 439.435,Z 265.377,A -85,B 0,C 180,E1 -8983.654,E2 -8983.654} C_VEL
LIN {X 0,Y 439.458,Z 265.371,A -85,B 0,C 180,E1 -8987.063,E2 -8987.063} C_VEL
LIN {X 0,Y 439.494,Z 265.367,A -85,B 0,C 180,E1 -8990.799,E2 -8990.799} C_VEL
LIN {X 0,Y 439.613,Z 265.352,A -85,B 0,C 180,E1 -8993.576,E2 -8993.576} C_VEL
LIN {X 0,Y 439.652,Z 265.347,A -85,B 0,C 180,E1 -8997.252,E2 -8997.252} C_VEL
LIN {X 0,Y 439.759,Z 265.331,A -85,B 0,C 180,E1 -9000.001,E2 -9000.001} C_VEL
LIN {X 0,Y 439.652,Z 265.348,A -85,B 0,C 180,E1 -9002.75,E2 -9002.75} C_VEL
LIN {X 0,Y 439.615,Z 265.349,A -85,B 0,C 180,E1 -9006.426,E2 -9006.426} C_VEL
LIN {X 0,Y 439.497,Z 265.366,A -85,B 0,C 180,E1 -9009.203,E2 -9009.203} C_VEL
LIN {X 0,Y 439.462,Z 265.368,A -85,B 0,C 180,E1 -9012.939,E2 -9012.939} C_VEL
LIN {X 0,Y 439.444,Z 265.372,A -85,B 0,C 180,E1 -9016.35,E2 -9016.35} C_VEL
LIN {X 0,Y 439.4,Z 265.377,A -85,B 0,C 180,E1 -9019.627,E2 -9019.627} C_VEL
LIN {X 0,Y 439.363,Z 265.384,A -85,B 0,C 180,E1 -9022.576,E2 -9022.576} C_VEL
LIN {X 0,Y 439.403,Z 265.377,A -85,B 0,C 180,E1 -9025.586,E2 -9025.586} C_VEL
LIN {X 0,Y 439.415,Z 265.378,A -85,B 0,C 180,E1 -9028.674,E2 -9028.674} C_VEL
LIN {X 0,Y 439.368,Z 265.387,A -85,B 0,C 180,E1 -9032.031,E2 -9032.031} C_VEL
LIN {X 0,Y 439.392,Z 265.385,A -85,B 0,C 180,E1 -9035.341,E2 -9035.341} C_VEL
LIN {X 0,Y 439.377,Z 265.387,A -85,B 0,C 180,E1 -9038.596,E2 -9038.596} C_VEL
LIN {X 0,Y 439.424,Z 265.521,A -85,B 0,C 180,E1 -9040.222,E2 -9040.222} C_VEL
LIN {X 0,Y 440.251,Z 270.4,A -85,B 0,C 180,E1 -9043.349,E2 -9043.349} C_VEL
LIN {X 0,Y 441.087,Z 274.669,A -85,B 0,C 180,E1 -9045.808,E2 -9045.808} C_VEL
LIN {X 0,Y 441.578,Z 278.793,A -85,B 0,C 180,E1 -9048.053,E2 -9048.053} C_VEL
LIN {X 0,Y 441.397,Z 283.632,A -85,B 0,C 180,E1 -9050.441,E2 -9050.441} C_VEL
LIN {X 0,Y 440.931,Z 289.88,A -85,B 0,C 180,E1 -9053.34,E2 -9053.34} C_VEL
LIN {X 0,Y 440.489,Z 297.304,A -85,B 0,C 180,E1 -9056.603,E2 -9056.603} C_VEL
LIN {X 0,Y 440.129,Z 304.396,A -85,B 0,C 180,E1 -9059.574,E2 -9059.574} C_VEL
LIN {X 0,Y 439.831,Z 311.388,A -85,B 0,C 180,E1 -9062.395,E2 -9062.395} C_VEL
LIN {X 0,Y 439.467,Z 319.883,A -85,B 0,C 180,E1 -9065.721,E2 -9065.721} C_VEL
LIN {X 0,Y 439.379,Z 322.49,A -85,B 0,C 180,E1 -9066.727,E2 -9066.727} C_VEL
LIN {X 0,Y 443.554,Z 340.135,A -85,B 0,C 180,E1 -9067.359,E2 -9067.359} C_VEL
LIN {X 0,Y 446.861,Z 354.822,A -85,B 0,C 180,E1 -9068.047,E2 -9068.047} C_VEL
LIN {X 0,Y 446.189,Z 368.75,A -85,B 0,C 180,E1 -9068.678,E2 -9068.678} C_VEL
LIN {X 0,Y 445.309,Z 382.068,A -85,B 0,C 180,E1 -9069.443,E2 -9069.443} C_VEL
LIN {X 0,Y 444.283,Z 395.021,A -85,B 0,C 180,E1 -9070.358,E2 -9070.358} C_VEL
LIN {X 0,Y 443.222,Z 408.328,A -85,B 0,C 180,E1 -9071.511,E2 -9071.511} C_VEL
LIN {X 0,Y 442.303,Z 419.51,A -85,B 0,C 180,E1 -9072.667,E2 -9072.667} C_VEL
LIN {X 0,Y 441.304,Z 430.811,A -85,B 0,C 180,E1 -9074.056,E2 -9074.056} C_VEL
LIN {X 0,Y 440.379,Z 441.794,A -85,B 0,C 180,E1 -9075.679,E2 -9075.679} C_VEL
LIN {X 0,Y 439.613,Z 450.482,A -85,B 0,C 180,E1 -9077.213,E2 -9077.213} C_VEL
LIN {X 0,Y 439.23,Z 458.558,A -85,B 0,C 180,E1 -9078.931,E2 -9078.931} C_VEL
LIN {X 0,Y 438.734,Z 465.654,A -85,B 0,C 180,E1 -9080.783,E2 -9080.783} C_VEL
LIN {X 0,Y 438.508,Z 471.245,A -85,B 0,C 180,E1 -9082.634,E2 -9082.634} C_VEL
LIN {X 0,Y 438.4,Z 475.476,A -85,B 0,C 180,E1 -9084.481,E2 -9084.481} C_VEL
LIN {X 0,Y 438.249,Z 478.439,A -85,B 0,C 180,E1 -9086.323,E2 -9086.323} C_VEL
LIN {X 0,Y 438.272,Z 480.215,A -85,B 0,C 180,E1 -9088.163,E2 -9088.163} C_VEL
LIN {X 0,Y 438.204,Z 480.821,A -85,B 0,C 180,E1 -9090.001,E2 -9090.001} C_VEL
LIN {X 0,Y 438.272,Z 480.22,A -85,B 0,C 180,E1 -9091.838,E2 -9091.838} C_VEL
LIN {X 0,Y 438.248,Z 478.451,A -85,B 0,C 180,E1 -9093.678,E2 -9093.678} C_VEL
LIN {X 0,Y 438.388,Z 475.502,A -85,B 0,C 180,E1 -9095.52,E2 -9095.52} C_VEL
LIN {X 0,Y 438.509,Z 471.291,A -85,B 0,C 180,E1 -9097.367,E2 -9097.367} C_VEL
LIN {X 0,Y 438.734,Z 465.714,A -85,B 0,C 180,E1 -9099.218,E2 -9099.218} C_VEL
LIN {X 0,Y 439.229,Z 458.633,A -85,B 0,C 180,E1 -9101.071,E2 -9101.071} C_VEL
LIN {X 0,Y 439.688,Z 450.355,A -85,B 0,C 180,E1 -9102.83,E2 -9102.83} C_VEL
LIN {X 0,Y 440.39,Z 441.932,A -85,B 0,C 180,E1 -9104.322,E2 -9104.322} C_VEL
LIN {X 0,Y 441.295,Z 430.98,A -85,B 0,C 180,E1 -9105.946,E2 -9105.946} C_VEL
LIN {X 0,Y 442.273,Z 419.749,A -85,B 0,C 180,E1 -9107.331,E2 -9107.331} C_VEL
LIN {X 0,Y 443.319,Z 407.394,A -85,B 0,C 180,E1 -9108.606,E2 -9108.606} C_VEL
LIN {X 0,Y 444.414,Z 393.86,A -85,B 0,C 180,E1 -9109.757,E2 -9109.757} C_VEL
LIN {X 0,Y 445.424,Z 380.588,A -85,B 0,C 180,E1 -9110.674,E2 -9110.674} C_VEL
LIN {X 0,Y 446.448,Z 365.506,A -85,B 0,C 180,E1 -9111.502,E2 -9111.502} C_VEL
LIN {X 0,Y 446.81,Z 354.441,A -85,B 0,C 180,E1 -9111.986,E2 -9111.986} C_VEL
LIN {X 0,Y 443.473,Z 339.723,A -85,B 0,C 180,E1 -9112.668,E2 -9112.668} C_VEL
LIN {X 0,Y 439.407,Z 323.048,A -85,B 0,C 180,E1 -9113.276,E2 -9113.276} C_VEL
LIN {X 0,Y 439.716,Z 316.016,A -85,B 0,C 180,E1 -9116.032,E2 -9116.032} C_VEL
LIN {X 0,Y 440.083,Z 308.297,A -85,B 0,C 180,E1 -9119.149,E2 -9119.149} C_VEL
LIN {X 0,Y 440.417,Z 300.847,A -85,B 0,C 180,E1 -9122.247,E2 -9122.247} C_VEL
LIN {X 0,Y 440.822,Z 294.409,A -85,B 0,C 180,E1 -9125.027,E2 -9125.027} C_VEL
LIN {X 0,Y 441.239,Z 288.135,A -85,B 0,C 180,E1 -9127.824,E2 -9127.824} C_VEL
LIN {X 0,Y 441.617,Z 283.049,A -85,B 0,C 180,E1 -9130.192,E2 -9130.192} C_VEL
LIN {X 0,Y 441.678,Z 279.465,A -85,B 0,C 180,E1 -9131.937,E2 -9131.937} C_VEL
LIN {X 0,Y 441.067,Z 274.497,A -85,B 0,C 180,E1 -9134.516,E2 -9134.516} C_VEL
LIN {X 0,Y 439.982,Z 268.53,A -85,B 0,C 180,E1 -9137.864,E2 -9137.864} C_VEL
LIN {X 0,Y 439.418,Z 265.377,A -85,B 0,C 180,E1 -9139.778,E2 -9139.778} C_VEL
LIN {X 0,Y 439.354,Z 265.383,A -85,B 0,C 180,E1 -9143.113,E2 -9143.113} C_VEL
LIN {X 0,Y 439.401,Z 265.377,A -85,B 0,C 180,E1 -9146.276,E2 -9146.276} C_VEL
LIN {X 0,Y 439.386,Z 265.377,A -85,B 0,C 180,E1 -9149.739,E2 -9149.739} C_VEL
LIN {X 0,Y 439.447,Z 265.372,A -85,B 0,C 180,E1 -9152.367,E2 -9152.367} C_VEL
LIN {X 0,Y 439.421,Z 265.372,A -85,B 0,C 180,E1 -9155.735,E2 -9155.735} C_VEL
LIN {X 0,Y 439.394,Z 265.376,A -85,B 0,C 180,E1 -9159.397,E2 -9159.397} C_VEL
LIN {X 0,Y 439.437,Z 265.373,A -85,B 0,C 180,E1 -9162.309,E2 -9162.309} C_VEL
LIN {X 0,Y 439.453,Z 265.37,A -85,B 0,C 180,E1 -9165.173,E2 -9165.173} C_VEL
LIN {X 0,Y 439.489,Z 265.366,A -85,B 0,C 180,E1 -9168.001,E2 -9168.001} C_VEL
LIN {X 0,Y 439.538,Z 265.358,A -85,B 0,C 180,E1 -9171.725,E2 -9171.725} C_VEL
LIN {X 0,Y 439.614,Z 265.352,A -85,B 0,C 180,E1 -9174.495,E2 -9174.495} C_VEL
LIN {X 0,Y 439.639,Z 265.349,A -85,B 0,C 180,E1 -9178.167,E2 -9178.167} C_VEL
LIN {X 0,Y 439.768,Z 265.332,A -85,B 0,C 180,E1 -9179.999,E2 -9179.999} C_VEL
LIN {X 0,Y 439.643,Z 265.348,A -85,B 0,C 180,E1 -9182.748,E2 -9182.748} C_VEL
LIN {X 0,Y 439.621,Z 265.352,A -85,B 0,C 180,E1 -9186.424,E2 -9186.424} C_VEL
LIN {X 0,Y 439.503,Z 265.362,A -85,B 0,C 180,E1 -9189.2,E2 -9189.2} C_VEL
LIN {X 0,Y 439.468,Z 265.367,A -85,B 0,C 180,E1 -9192.936,E2 -9192.936} C_VEL
LIN {X 0,Y 439.449,Z 265.373,A -85,B 0,C 180,E1 -9196.348,E2 -9196.348} C_VEL
LIN {X 0,Y 439.403,Z 265.377,A -85,B 0,C 180,E1 -9199.625,E2 -9199.625} C_VEL
LIN {X 0,Y 439.366,Z 265.382,A -85,B 0,C 180,E1 -9202.574,E2 -9202.574} C_VEL
LIN {X 0,Y 439.405,Z 265.377,A -85,B 0,C 180,E1 -9205.583,E2 -9205.583} C_VEL
LIN {X 0,Y 439.416,Z 265.374,A -85,B 0,C 180,E1 -9208.672,E2 -9208.672} C_VEL
LIN {X 0,Y 439.368,Z 265.383,A -85,B 0,C 180,E1 -9212.029,E2 -9212.029} C_VEL
LIN {X 0,Y 439.394,Z 265.377,A -85,B 0,C 180,E1 -9215.339,E2 -9215.339} C_VEL
LIN {X 0,Y 439.387,Z 265.378,A -85,B 0,C 180,E1 -9218.593,E2 -9218.593} C_VEL
LIN {X 0,Y 439.385,Z 265.378,A -85,B 0,C 180,E1 -9221.256,E2 -9221.256} C_VEL
LIN {X 0,Y 439.402,Z 265.375,A -85,B 0,C 180,E1 -9224.727,E2 -9224.727} C_VEL
LIN {X 0,Y 439.407,Z 265.378,A -85,B 0,C 180,E1 -9227.796,E2 -9227.796} C_VEL
LIN {X 0,Y 439.443,Z 265.372,A -85,B 0,C 180,E1 -9230.229,E2 -9230.229} C_VEL
LIN {X 0,Y 439.371,Z 265.383,A -85,B 0,C 180,E1 -9233.712,E2 -9233.712} C_VEL
LIN {X 0,Y 439.365,Z 265.381,A -85,B 0,C 180,E1 -9237.053,E2 -9237.053} C_VEL
LIN {X 0,Y 439.389,Z 265.378,A -85,B 0,C 180,E1 -9240.274,E2 -9240.274} C_VEL
LIN {X 0,Y 439.425,Z 265.376,A -85,B 0,C 180,E1 -9243.587,E2 -9243.587} C_VEL
LIN {X 0,Y 439.378,Z 265.377,A -85,B 0,C 180,E1 -9246.428,E2 -9246.428} C_VEL
LIN {X 0,Y 439.38,Z 265.382,A -85,B 0,C 180,E1 -9249.396,E2 -9249.396} C_VEL
LIN {X 0,Y 439.422,Z 265.373,A -85,B 0,C 180,E1 -9252.309,E2 -9252.309} C_VEL
LIN {X 0,Y 439.439,Z 265.374,A -85,B 0,C 180,E1 -9255.173,E2 -9255.173} C_VEL
LIN {X 0,Y 439.498,Z 265.364,A -85,B 0,C 180,E1 -9258.001,E2 -9258.001} C_VEL
LIN {X 0,Y 439.538,Z 265.36,A -85,B 0,C 180,E1 -9261.725,E2 -9261.725} C_VEL
LIN {X 0,Y 439.597,Z 265.35,A -85,B 0,C 180,E1 -9264.495,E2 -9264.495} C_VEL
LIN {X 0,Y 439.241,Z 265.4,A -85,B 0,C 180,E1 -9268.166,E2 -9268.166} C_VEL
LIN {X 0,Y 439.424,Z 265.686,A -85,B 0,C 180,E1 -9269.083,E2 -9269.083} C_VEL
LIN {X 0,Y 439.031,Z 267.396,A -85,B 0,C 180,E1 -9270.976,E2 -9270.976} C_VEL
LIN {X 0,Y 438.219,Z 268.16,A -85,B 0,C 180,E1 -9271.733,E2 -9271.733} C_VEL
LIN {X 0,Y 435.335,Z 269.588,A -85,B 0,C 180,E1 -9272.963,E2 -9272.963} C_VEL
LIN {X 0,Y 432.973,Z 270.74,A -85,B 0,C 180,E1 -9273.954,E2 -9273.954} C_VEL
LIN {X 0,Y 431.949,Z 271.538,A -85,B 0,C 180,E1 -9274.721,E2 -9274.721} C_VEL
LIN {X 0,Y 431.854,Z 271.778,A -85,B 0,C 180,E1 -9274.981,E2 -9274.981} C_VEL
LIN {X 0,Y 431.786,Z 274.036,A -85,B 0,C 180,E1 -9277.481,E2 -9277.481} C_VEL
LIN {X 0,Y 431.701,Z 275.859,A -85,B 0,C 180,E1 -9279.478,E2 -9279.478} C_VEL
LIN {X 0,Y 434.226,Z 283.424,A -85,B 0,C 180,E1 -9279.798,E2 -9279.798} C_VEL
LIN {X 0,Y 438.687,Z 296.793,A -85,B 0,C 180,E1 -9280.464,E2 -9280.464} C_VEL
LIN {X 0,Y 440.623,Z 304.033,A -85,B 0,C 180,E1 -9280.86,E2 -9280.86} C_VEL
LIN {X 0,Y 439.762,Z 319.131,A -85,B 0,C 180,E1 -9281.571,E2 -9281.571} C_VEL
LIN {X 0,Y 438.814,Z 334.036,A -85,B 0,C 180,E1 -9282.494,E2 -9282.494} C_VEL
LIN {X 0,Y 437.81,Z 347.93,A -85,B 0,C 180,E1 -9283.577,E2 -9283.577} C_VEL
LIN {X 0,Y 436.647,Z 361.239,A -85,B 0,C 180,E1 -9284.851,E2 -9284.851} C_VEL
LIN {X 0,Y 435.673,Z 372.511,A -85,B 0,C 180,E1 -9286.156,E2 -9286.156} C_VEL
LIN {X 0,Y 434.668,Z 383.187,A -85,B 0,C 180,E1 -9287.629,E2 -9287.629} C_VEL
LIN {X 0,Y 433.734,Z 392.442,A -85,B 0,C 180,E1 -9289.154,E2 -9289.154} C_VEL
LIN {X 0,Y 432.999,Z 401.34,A -85,B 0,C 180,E1 -9290.92,E2 -9290.92} C_VEL
LIN {X 0,Y 432.461,Z 407.944,A -85,B 0,C 180,E1 -9292.51,E2 -9292.51} C_VEL
LIN {X 0,Y 431.929,Z 414.161,A -85,B 0,C 180,E1 -9294.334,E2 -9294.334} C_VEL
LIN {X 0,Y 431.686,Z 418.842,A -85,B 0,C 180,E1 -9296.076,E2 -9296.076} C_VEL
LIN {X 0,Y 431.566,Z 421.112,A -85,B 0,C 180,E1 -9297.127,E2 -9297.127} C_VEL
LIN {X 0,Y 431.259,Z 424.558,A -85,B 0,C 180,E1 -9299.267,E2 -9299.267} C_VEL
LIN {X 0,Y 431.197,Z 425.713,A -85,B 0,C 180,E1 -9300.348,E2 -9300.348} C_VEL
LIN {X 0,Y 431.155,Z 426.799,A -85,B 0,C 180,E1 -9302.049,E2 -9302.049} C_VEL
LIN {X 0,Y 431.151,Z 426.885,A -85,B 0,C 180,E1 -9303.767,E2 -9303.767} C_VEL
LIN {X 0,Y 431.211,Z 425.692,A -85,B 0,C 180,E1 -9305.925,E2 -9305.925} C_VEL
LIN {X 0,Y 431.3,Z 424.442,A -85,B 0,C 180,E1 -9307.078,E2 -9307.078} C_VEL
LIN {X 0,Y 431.524,Z 422.097,A -85,B 0,C 180,E1 -9308.581,E2 -9308.581} C_VEL
LIN {X 0,Y 431.791,Z 417.693,A -85,B 0,C 180,E1 -9310.62,E2 -9310.62} C_VEL
LIN {X 0,Y 432.149,Z 412.571,A -85,B 0,C 180,E1 -9312.408,E2 -9312.408} C_VEL
LIN {X 0,Y 432.685,Z 405.688,A -85,B 0,C 180,E1 -9314.301,E2 -9314.301} C_VEL
LIN {X 0,Y 433.415,Z 398.184,A -85,B 0,C 180,E1 -9315.976,E2 -9315.976} C_VEL
LIN {X 0,Y 434.206,Z 389.611,A -85,B 0,C 180,E1 -9317.565,E2 -9317.565} C_VEL
LIN {X 0,Y 435.147,Z 379.585,A -85,B 0,C 180,E1 -9319.116,E2 -9319.116} C_VEL
LIN {X 0,Y 436.133,Z 369.618,A -85,B 0,C 180,E1 -9320.408,E2 -9320.408} C_VEL
LIN {X 0,Y 437.246,Z 357.798,A -85,B 0,C 180,E1 -9321.7,E2 -9321.7} C_VEL
LIN {X 0,Y 438.344,Z 344.74,A -85,B 0,C 180,E1 -9322.883,E2 -9322.883} C_VEL
LIN {X 0,Y 439.295,Z 331.984,A -85,B 0,C 180,E1 -9323.829,E2 -9323.829} C_VEL
LIN {X 0,Y 440.194,Z 318.168,A -85,B 0,C 180,E1 -9324.654,E2 -9324.654} C_VEL
LIN {X 0,Y 440.774,Z 303.98,A -85,B 0,C 180,E1 -9325.319,E2 -9325.319} C_VEL
LIN {X 0,Y 436.571,Z 290.612,A -85,B 0,C 180,E1 -9326.055,E2 -9326.055} C_VEL
LIN {X 0,Y 431.904,Z 277.948,A -85,B 0,C 180,E1 -9326.656,E2 -9326.656} C_VEL
LIN {X 0,Y 431.814,Z 277.383,A -85,B 0,C 180,E1 -9326.683,E2 -9326.683} C_VEL
LIN {X 0,Y 431.893,Z 274.839,A -85,B 0,C 180,E1 -9329.707,E2 -9329.707} C_VEL
LIN {X 0,Y 431.948,Z 272.189,A -85,B 0,C 180,E1 -9332.9,E2 -9332.9} C_VEL
LIN {X 0,Y 432.102,Z 269.639,A -85,B 0,C 180,E1 -9336.009,E2 -9336.009} C_VEL
LIN {X 0,Y 432.15,Z 267.186,A -85,B 0,C 180,E1 -9339.037,E2 -9339.037} C_VEL
LIN {X 0,Y 432.177,Z 266.392,A -85,B 0,C 180,E1 -9340.033,E2 -9340.033} C_VEL
LIN {X 0,Y 432.34,Z 266.262,A -85,B 0,C 180,E1 -9342.987,E2 -9342.987} C_VEL
LIN {X 0,Y 432.367,Z 266.255,A -85,B 0,C 180,E1 -9345.889,E2 -9345.889} C_VEL
LIN {X 0,Y 432.387,Z 266.253,A -85,B 0,C 180,E1 -9348.754,E2 -9348.754} C_VEL
LIN {X 0,Y 432.58,Z 266.227,A -85,B 0,C 180,E1 -9352.322,E2 -9352.322} C_VEL
LIN {X 0,Y 432.593,Z 266.226,A -85,B 0,C 180,E1 -9354.407,E2 -9354.407} C_VEL
LIN {X 0,Y 432.601,Z 266.224,A -85,B 0,C 180,E1 -9358.139,E2 -9358.139} C_VEL
LIN {X 0,Y 432.729,Z 266.207,A -85,B 0,C 180,E1 -9360.001,E2 -9360.001} C_VEL
LIN {X 0,Y 432.601,Z 266.226,A -85,B 0,C 180,E1 -9362.795,E2 -9362.795} C_VEL
LIN {X 0,Y 432.569,Z 266.227,A -85,B 0,C 180,E1 -9366.531,E2 -9366.531} C_VEL
LIN {X 0,Y 432.44,Z 266.245,A -85,B 0,C 180,E1 -9369.354,E2 -9369.354} C_VEL
LIN {X 0,Y 432.427,Z 266.244,A -85,B 0,C 180,E1 -9372.804,E2 -9372.804} C_VEL
LIN {X 0,Y 432.409,Z 266.248,A -85,B 0,C 180,E1 -9376.48,E2 -9376.48} C_VEL
LIN {X 0,Y 432.336,Z 266.257,A -85,B 0,C 180,E1 -9379.961,E2 -9379.961} C_VEL
LIN {X 0,Y 432.317,Z 266.26,A -85,B 0,C 180,E1 -9382.965,E2 -9382.965} C_VEL
LIN {X 0,Y 432.362,Z 266.256,A -85,B 0,C 180,E1 -9386.033,E2 -9386.033} C_VEL
LIN {X 0,Y 432.341,Z 266.259,A -85,B 0,C 180,E1 -9389.188,E2 -9389.188} C_VEL
LIN {X 0,Y 432.321,Z 266.264,A -85,B 0,C 180,E1 -9392.444,E2 -9392.444} C_VEL
LIN {X 0,Y 432.342,Z 266.264,A -85,B 0,C 180,E1 -9395.633,E2 -9395.633} C_VEL
LIN {X 0,Y 432.345,Z 266.26,A -85,B 0,C 180,E1 -9399.344,E2 -9399.344} C_VEL
LIN {X 0,Y 432.419,Z 266.456,A -85,B 0,C 180,E1 -9399.776,E2 -9399.776} C_VEL
LIN {X 0,Y 433.24,Z 271.49,A -85,B 0,C 180,E1 -9403.116,E2 -9403.116} C_VEL
LIN {X 0,Y 434.164,Z 276.21,A -85,B 0,C 180,E1 -9405.889,E2 -9405.889} C_VEL
LIN {X 0,Y 434.617,Z 280.153,A -85,B 0,C 180,E1 -9408.061,E2 -9408.061} C_VEL
LIN {X 0,Y 434.32,Z 285.973,A -85,B 0,C 180,E1 -9410.962,E2 -9410.962} C_VEL
LIN {X 0,Y 433.781,Z 292.724,A -85,B 0,C 180,E1 -9414.105,E2 -9414.105} C_VEL
LIN {X 0,Y 433.412,Z 299.419,A -85,B 0,C 180,E1 -9417.069,E2 -9417.069} C_VEL
LIN {X 0,Y 433.017,Z 307.11,A -85,B 0,C 180,E1 -9420.329,E2 -9420.329} C_VEL
LIN {X 0,Y 432.696,Z 314.358,A -85,B 0,C 180,E1 -9423.295,E2 -9423.295} C_VEL
LIN {X 0,Y 432.39,Z 322.24,A -85,B 0,C 180,E1 -9426.336,E2 -9426.336} C_VEL
LIN {X 0,Y 436.392,Z 339.047,A -85,B 0,C 180,E1 -9426.95,E2 -9426.95} C_VEL
LIN {X 0,Y 439.911,Z 354.808,A -85,B 0,C 180,E1 -9427.702,E2 -9427.702} C_VEL
LIN {X 0,Y 440.025,Z 359.619,A -85,B 0,C 180,E1 -9427.925,E2 -9427.925} C_VEL
LIN {X 0,Y 439.193,Z 373.955,A -85,B 0,C 180,E1 -9428.652,E2 -9428.652} C_VEL
LIN {X 0,Y 438.011,Z 388.35,A -85,B 0,C 180,E1 -9429.576,E2 -9429.576} C_VEL
LIN {X 0,Y 436.931,Z 401.49,A -85,B 0,C 180,E1 -9430.626,E2 -9430.626} C_VEL
LIN {X 0,Y 435.893,Z 413.642,A -85,B 0,C 180,E1 -9431.798,E2 -9431.798} C_VEL
LIN {X 0,Y 434.925,Z 424.915,A -85,B 0,C 180,E1 -9433.091,E2 -9433.091} C_VEL
LIN {X 0,Y 433.923,Z 435.283,A -85,B 0,C 180,E1 -9434.501,E2 -9434.501} C_VEL
LIN {X 0,Y 433.044,Z 445.443,A -85,B 0,C 180,E1 -9436.151,E2 -9436.151} C_VEL
LIN {X 0,Y 432.406,Z 453.893,A -85,B 0,C 180,E1 -9437.803,E2 -9437.803} C_VEL
LIN {X 0,Y 432.026,Z 459.994,A -85,B 0,C 180,E1 -9439.218,E2 -9439.218} C_VEL
LIN {X 0,Y 431.587,Z 466.711,A -85,B 0,C 180,E1 -9441.101,E2 -9441.101} C_VEL
LIN {X 0,Y 431.412,Z 471.98,A -85,B 0,C 180,E1 -9442.983,E2 -9442.983} C_VEL
LIN {X 0,Y 431.31,Z 475.026,A -85,B 0,C 180,E1 -9444.39,E2 -9444.39} C_VEL
LIN {X 0,Y 431.159,Z 477.994,A -85,B 0,C 180,E1 -9446.262,E2 -9446.262} C_VEL
LIN {X 0,Y 431.263,Z 479.037,A -85,B 0,C 180,E1 -9447.198,E2 -9447.198} C_VEL
LIN {X 0,Y 431.146,Z 480.226,A -85,B 0,C 180,E1 -9449.067,E2 -9449.067} C_VEL
LIN {X 0,Y 431.146,Z 480.233,A -85,B 0,C 180,E1 -9450.935,E2 -9450.935} C_VEL
LIN {X 0,Y 431.263,Z 479.053,A -85,B 0,C 180,E1 -9452.803,E2 -9452.803} C_VEL
LIN {X 0,Y 431.235,Z 476.696,A -85,B 0,C 180,E1 -9454.675,E2 -9454.675} C_VEL
LIN {X 0,Y 431.374,Z 473.128,A -85,B 0,C 180,E1 -9456.549,E2 -9456.549} C_VEL
LIN {X 0,Y 431.52,Z 468.248,A -85,B 0,C 180,E1 -9458.429,E2 -9458.429} C_VEL
LIN {X 0,Y 431.836,Z 461.936,A -85,B 0,C 180,E1 -9460.313,E2 -9460.313} C_VEL
LIN {X 0,Y 432.368,Z 455.125,A -85,B 0,C 180,E1 -9461.962,E2 -9461.962} C_VEL
LIN {X 0,Y 432.951,Z 446.887,A -85,B 0,C 180,E1 -9463.614,E2 -9463.614} C_VEL
LIN {X 0,Y 433.826,Z 437.029,A -85,B 0,C 180,E1 -9465.264,E2 -9465.264} C_VEL
LIN {X 0,Y 434.72,Z 426.956,A -85,B 0,C 180,E1 -9466.677,E2 -9466.677} C_VEL
LIN {X 0,Y 435.812,Z 415.011,A -85,B 0,C 180,E1 -9468.086,E2 -9468.086} C_VEL
LIN {X 0,Y 436.816,Z 403.116,A -85,B 0,C 180,E1 -9469.259,E2 -9469.259} C_VEL
LIN {X 0,Y 437.889,Z 390.289,A -85,B 0,C 180,E1 -9470.309,E2 -9470.309} C_VEL
LIN {X 0,Y 439.05,Z 376.328,A -85,B 0,C 180,E1 -9471.234,E2 -9471.234} C_VEL
LIN {X 0,Y 439.964,Z 361.993,A -85,B 0,C 180,E1 -9471.987,E2 -9471.987} C_VEL
LIN {X 0,Y 440.102,Z 355.456,A -85,B 0,C 180,E1 -9472.281,E2 -9472.281} C_VEL
LIN {X 0,Y 436.704,Z 340.555,A -85,B 0,C 180,E1 -9473.006,E2 -9473.006} C_VEL
LIN {X 0,Y 432.805,Z 324.856,A -85,B 0,C 180,E1 -9473.601,E2 -9473.601} C_VEL
LIN {X 0,Y 432.385,Z 322.623,A -85,B 0,C 180,E1 -9473.676,E2 -9473.676} C_VEL
LIN {X 0,Y 432.79,Z 314.26,A -85,B 0,C 180,E1 -9477.045,E2 -9477.045} C_VEL
LIN {X 0,Y 433.158,Z 306.651,A -85,B 0,C 180,E1 -9480.198,E2 -9480.198} C_VEL
LIN {X 0,Y 433.576,Z 299.1,A -85,B 0,C 180,E1 -9483.444,E2 -9483.444} C_VEL
LIN {X 0,Y 434.11,Z 291.598,A -85,B 0,C 180,E1 -9486.8,E2 -9486.8} C_VEL
LIN {X 0,Y 434.661,Z 284.132,A -85,B 0,C 180,E1 -9490.298,E2 -9490.298} C_VEL
LIN {X 0,Y 434.727,Z 280.789,A -85,B 0,C 180,E1 -9491.955,E2 -9491.955} C_VEL
LIN {X 0,Y 434.098,Z 275.837,A -85,B 0,C 180,E1 -9494.572,E2 -9494.572} C_VEL
LIN {X 0,Y 433.111,Z 270.372,A -85,B 0,C 180,E1 -9497.668,E2 -9497.668} C_VEL
LIN {X 0,Y 432.407,Z 266.25,A -85,B 0,C 180,E1 -9500.228,E2 -9500.228} C_VEL
LIN {X 0,Y 432.312,Z 266.26,A -85,B 0,C 180,E1 -9503.022,E2 -9503.022} C_VEL
LIN {X 0,Y 432.363,Z 266.254,A -85,B 0,C 180,E1 -9505.997,E2 -9505.997} C_VEL
LIN {X 0,Y 432.353,Z 266.254,A -85,B 0,C 180,E1 -9509.489,E2 -9509.489} C_VEL
LIN {X 0,Y 432.397,Z 266.252,A -85,B 0,C 180,E1 -9512.928,E2 -9512.928} C_VEL
LIN {X 0,Y 432.377,Z 266.25,A -85,B 0,C 180,E1 -9516.023,E2 -9516.023} C_VEL
LIN {X 0,Y 432.356,Z 266.255,A -85,B 0,C 180,E1 -9519.046,E2 -9519.046} C_VEL
LIN {X 0,Y 432.384,Z 266.25,A -85,B 0,C 180,E1 -9522.011,E2 -9522.011} C_VEL
LIN {X 0,Y 432.401,Z 266.25,A -85,B 0,C 180,E1 -9524.926,E2 -9524.926} C_VEL
LIN {X 0,Y 432.464,Z 266.24,A -85,B 0,C 180,E1 -9527.803,E2 -9527.803} C_VEL
LIN {X 0,Y 432.488,Z 266.236,A -85,B 0,C 180,E1 -9531.589,E2 -9531.589} C_VEL
LIN {X 0,Y 432.59,Z 266.227,A -85,B 0,C 180,E1 -9534.405,E2 -9534.405} C_VEL
LIN {X 0,Y 432.609,Z 266.224,A -85,B 0,C 180,E1 -9538.137,E2 -9538.137} C_VEL
LIN {X 0,Y 432.738,Z 266.207,A -85,B 0,C 180,E1 -9539.999,E2 -9539.999} C_VEL
LIN {X 0,Y 432.595,Z 266.226,A -85,B 0,C 180,E1 -9542.793,E2 -9542.793} C_VEL
LIN {X 0,Y 432.576,Z 266.229,A -85,B 0,C 180,E1 -9546.529,E2 -9546.529} C_VEL
LIN {X 0,Y 432.446,Z 266.241,A -85,B 0,C 180,E1 -9549.352,E2 -9549.352} C_VEL
LIN {X 0,Y 432.433,Z 266.244,A -85,B 0,C 180,E1 -9552.802,E2 -9552.802} C_VEL
LIN {X 0,Y 432.414,Z 266.249,A -85,B 0,C 180,E1 -9556.478,E2 -9556.478} C_VEL
LIN {X 0,Y 432.34,Z 266.258,A -85,B 0,C 180,E1 -9559.959,E2 -9559.959} C_VEL
LIN {X 0,Y 432.32,Z 266.257,A -85,B 0,C 180,E1 -9562.963,E2 -9562.963} C_VEL
LIN {X 0,Y 432.364,Z 266.256,A -85,B 0,C 180,E1 -9566.031,E2 -9566.031} C_VEL
LIN {X 0,Y 432.342,Z 266.254,A -85,B 0,C 180,E1 -9569.186,E2 -9569.186} C_VEL
LIN {X 0,Y 432.321,Z 266.259,A -85,B 0,C 180,E1 -9572.442,E2 -9572.442} C_VEL
LIN {X 0,Y 432.343,Z 266.257,A -85,B 0,C 180,E1 -9575.631,E2 -9575.631} C_VEL
LIN {X 0,Y 432.349,Z 266.254,A -85,B 0,C 180,E1 -9578.715,E2 -9578.715} C_VEL
LIN {X 0,Y 432.331,Z 266.26,A -85,B 0,C 180,E1 -9581.795,E2 -9581.795} C_VEL
LIN {X 0,Y 432.373,Z 266.254,A -85,B 0,C 180,E1 -9585.657,E2 -9585.657} C_VEL
LIN {X 0,Y 432.368,Z 266.252,A -85,B 0,C 180,E1 -9588.391,E2 -9588.391} C_VEL
LIN {X 0,Y 432.345,Z 266.258,A -85,B 0,C 180,E1 -9591.85,E2 -9591.85} C_VEL
LIN {X 0,Y 432.334,Z 266.258,A -85,B 0,C 180,E1 -9595.322,E2 -9595.322} C_VEL
LIN {X 0,Y 432.317,Z 266.258,A -85,B 0,C 180,E1 -9598.653,E2 -9598.653} C_VEL
LIN {X 0,Y 432.373,Z 266.254,A -85,B 0,C 180,E1 -9601.368,E2 -9601.368} C_VEL
LIN {X 0,Y 432.356,Z 266.255,A -85,B 0,C 180,E1 -9603.966,E2 -9603.966} C_VEL
LIN {X 0,Y 432.31,Z 266.259,A -85,B 0,C 180,E1 -9607.035,E2 -9607.035} C_VEL
LIN {X 0,Y 432.377,Z 266.25,A -85,B 0,C 180,E1 -9610.514,E2 -9610.514} C_VEL
LIN {X 0,Y 432.421,Z 266.246,A -85,B 0,C 180,E1 -9613.96,E2 -9613.96} C_VEL
LIN {X 0,Y 432.471,Z 266.241,A -85,B 0,C 180,E1 -9617.803,E2 -9617.803} C_VEL
LIN {X 0,Y 432.482,Z 266.241,A -85,B 0,C 180,E1 -9621.59,E2 -9621.59} C_VEL
LIN {X 0,Y 432.575,Z 266.225,A -85,B 0,C 180,E1 -9624.405,E2 -9624.405} C_VEL
LIN {X 0,Y 432.39,Z 266.507,A -85,B 0,C 180,E1 -9629.068,E2 -9629.068} C_VEL
LIN {X 0,Y 431.865,Z 270.659,A -85,B 0,C 180,E1 -9633.732,E2 -9633.732} C_VEL
LIN {X 0,Y 431.854,Z 271.778,A -85,B 0,C 180,E1 -9634.981,E2 -9634.981} C_VEL
LIN {X 0,Y 431.141,Z 272.549,A -85,B 0,C 180,E1 -9635.753,E2 -9635.753} C_VEL
LIN {X 0,Y 428.221,Z 274.003,A -85,B 0,C 180,E1 -9637.004,E2 -9637.004} C_VEL
LIN {X 0,Y 425.778,Z 275.181,A -85,B 0,C 180,E1 -9638.012,E2 -9638.012} C_VEL
LIN {X 0,Y 424.742,Z 276.002,A -85,B 0,C 180,E1 -9638.794,E2 -9638.794} C_VEL
LIN {X 0,Y 424.665,Z 276.252,A -85,B 0,C 180,E1 -9639.059,E2 -9639.059} C_VEL
LIN {X 0,Y 426.324,Z 281.376,A -85,B 0,C 180,E1 -9639.295,E2 -9639.295} C_VEL
LIN {X 0,Y 431.33,Z 295.851,A -85,B 0,C 180,E1 -9640.02,E2 -9640.02} C_VEL
LIN {X 0,Y 433.721,Z 304.37,A -85,B 0,C 180,E1 -9640.494,E2 -9640.494} C_VEL
LIN {X 0,Y 433.879,Z 308.155,A -85,B 0,C 180,E1 -9640.677,E2 -9640.677} C_VEL
LIN {X 0,Y 433.002,Z 322.491,A -85,B 0,C 180,E1 -9641.408,E2 -9641.408} C_VEL
LIN {X 0,Y 432.027,Z 336.218,A -85,B 0,C 180,E1 -9642.303,E2 -9642.303} C_VEL
LIN {X 0,Y 431.055,Z 348.805,A -85,B 0,C 180,E1 -9643.314,E2 -9643.314} C_VEL
LIN {X 0,Y 429.933,Z 361.305,A -85,B 0,C 180,E1 -9644.528,E2 -9644.528} C_VEL
LIN {X 0,Y 428.824,Z 373.256,A -85,B 0,C 180,E1 -9645.932,E2 -9645.932} C_VEL
LIN {X 0,Y 427.893,Z 382.319,A -85,B 0,C 180,E1 -9647.195,E2 -9647.195} C_VEL
LIN {X 0,Y 426.942,Z 391.667,A -85,B 0,C 180,E1 -9648.722,E2 -9648.722} C_VEL
LIN {X 0,Y 426.139,Z 400.771,A -85,B 0,C 180,E1 -9650.515,E2 -9650.515} C_VEL
LIN {X 0,Y 425.456,Z 408.321,A -85,B 0,C 180,E1 -9652.329,E2 -9652.329} C_VEL
LIN {X 0,Y 424.965,Z 413.718,A -85,B 0,C 180,E1 -9653.901,E2 -9653.901} C_VEL
LIN {X 0,Y 424.675,Z 418.121,A -85,B 0,C 180,E1 -9655.484,E2 -9655.484} C_VEL
LIN {X 0,Y 424.555,Z 420.763,A -85,B 0,C 180,E1 -9656.636,E2 -9656.636} C_VEL
LIN {X 0,Y 424.243,Z 424.368,A -85,B 0,C 180,E1 -9658.712,E2 -9658.712} C_VEL
LIN {X 0,Y 424.081,Z 426.664,A -85,B 0,C 180,E1 -9660.913,E2 -9660.913} C_VEL
LIN {X 0,Y 424.068,Z 427.291,A -85,B 0,C 180,E1 -9662.308,E2 -9662.308} C_VEL
LIN {X 0,Y 424.059,Z 427.196,A -85,B 0,C 180,E1 -9664.296,E2 -9664.296} C_VEL
LIN {X 0,Y 424.123,Z 426.348,A -85,B 0,C 180,E1 -9665.715,E2 -9665.715} C_VEL
LIN {X 0,Y 424.315,Z 423.979,A -85,B 0,C 180,E1 -9667.794,E2 -9667.794} C_VEL
LIN {X 0,Y 424.546,Z 420.802,A -85,B 0,C 180,E1 -9669.592,E2 -9669.592} C_VEL
LIN {X 0,Y 424.885,Z 416.425,A -85,B 0,C 180,E1 -9671.424,E2 -9671.424} C_VEL
LIN {X 0,Y 425.36,Z 410.379,A -85,B 0,C 180,E1 -9673.368,E2 -9673.368} C_VEL
LIN {X 0,Y 426.082,Z 403.306,A -85,B 0,C 180,E1 -9675.174,E2 -9675.174} C_VEL
LIN {X 0,Y 426.759,Z 395.683,A -85,B 0,C 180,E1 -9676.778,E2 -9676.778} C_VEL
LIN {X 0,Y 427.683,Z 386.534,A -85,B 0,C 180,E1 -9678.389,E2 -9678.389} C_VEL
LIN {X 0,Y 428.665,Z 376.693,A -85,B 0,C 180,E1 -9679.844,E2 -9679.844} C_VEL
LIN {X 0,Y 429.884,Z 364.83,A -85,B 0,C 180,E1 -9681.306,E2 -9681.306} C_VEL
LIN {X 0,Y 431.1,Z 352.023,A -85,B 0,C 180,E1 -9682.61,E2 -9682.61} C_VEL
LIN {X 0,Y 432.162,Z 339.347,A -85,B 0,C 180,E1 -9683.672,E2 -9683.672} C_VEL
LIN {X 0,Y 433.238,Z 325.436,A -85,B 0,C 180,E1 -9684.613,E2 -9684.613} C_VEL
LIN {X 0,Y 434.059,Z 311.261,A -85,B 0,C 180,E1 -9685.372,E2 -9685.372} C_VEL
LIN {X 0,Y 434.184,Z 305.576,A -85,B 0,C 180,E1 -9685.634,E2 -9685.634} C_VEL
LIN {X 0,Y 429.769,Z 291.605,A -85,B 0,C 180,E1 -9686.433,E2 -9686.433} C_VEL
LIN {X 0,Y 424.826,Z 278.096,A -85,B 0,C 180,E1 -9687.094,E2 -9687.094} C_VEL
LIN {X 0,Y 424.833,Z 275.276,A -85,B 0,C 180,E1 -9690.247,E2 -9690.247} C_VEL
LIN {X 0,Y 424.966,Z 272.616,A -85,B 0,C 180,E1 -9693.481,E2 -9693.481} C_VEL
LIN {X 0,Y 425.072,Z 270.097,A -85,B 0,C 180,E1 -9696.623,E2 -9696.623} C_VEL
LIN {X 0,Y 425.145,Z 267.66,A -85,B 0,C 180,E1 -9699.688,E2 -9699.688} C_VEL
LIN {X 0,Y 425.198,Z 267.149,A -85,B 0,C 180,E1 -9700.698,E2 -9700.698} C_VEL
LIN {X 0,Y 425.367,Z 267.13,A -85,B 0,C 180,E1 -9703.689,E2 -9703.689} C_VEL
LIN {X 0,Y 425.386,Z 267.123,A -85,B 0,C 180,E1 -9707.097,E2 -9707.097} C_VEL
LIN {X 0,Y 425.395,Z 267.124,A -85,B 0,C 180,E1 -9710.492,E2 -9710.492} C_VEL
LIN {X 0,Y 425.526,Z 267.107,A -85,B 0,C 180,E1 -9713.362,E2 -9713.362} C_VEL
LIN {X 0,Y 425.367,Z 267.127,A -85,B 0,C 180,E1 -9715.262,E2 -9715.262} C_VEL
LIN {X 0,Y 425.57,Z 267.1,A -85,B 0,C 180,E1 -9718.108,E2 -9718.108} C_VEL
LIN {X 0,Y 425.699,Z 267.083,A -85,B 0,C 180,E1 -9720.001,E2 -9720.001} C_VEL
LIN {X 0,Y 425.553,Z 267.103,A -85,B 0,C 180,E1 -9722.841,E2 -9722.841} C_VEL
LIN {X 0,Y 425.527,Z 267.105,A -85,B 0,C 180,E1 -9726.64,E2 -9726.64} C_VEL
LIN {X 0,Y 425.398,Z 267.122,A -85,B 0,C 180,E1 -9729.51,E2 -9729.51} C_VEL
LIN {X 0,Y 425.39,Z 267.121,A -85,B 0,C 180,E1 -9732.905,E2 -9732.905} C_VEL
LIN {X 0,Y 425.358,Z 267.126,A -85,B 0,C 180,E1 -9736.606,E2 -9736.606} C_VEL
LIN {X 0,Y 425.326,Z 267.129,A -85,B 0,C 180,E1 -9739.637,E2 -9739.637} C_VEL
LIN {X 0,Y 425.304,Z 267.132,A -85,B 0,C 180,E1 -9743.366,E2 -9743.366} C_VEL
LIN {X 0,Y 425.346,Z 267.128,A -85,B 0,C 180,E1 -9746.845,E2 -9746.845} C_VEL
LIN {X 0,Y 425.289,Z 267.139,A -85,B 0,C 180,E1 -9749.72,E2 -9749.72} C_VEL
LIN {X 0,Y 425.28,Z 267.144,A -85,B 0,C 180,E1 -9753.049,E2 -9753.049} C_VEL
LIN {X 0,Y 425.28,Z 267.145,A -85,B 0,C 180,E1 -9755.93,E2 -9755.93} C_VEL
LIN {X 0,Y 425.335,Z 267.3,A -85,B 0,C 180,E1 -9759.249,E2 -9759.249} C_VEL
LIN {X 0,Y 426.045,Z 271.4,A -85,B 0,C 180,E1 -9762.072,E2 -9762.072} C_VEL
LIN {X 0,Y 427.154,Z 277.24,A -85,B 0,C 180,E1 -9765.679,E2 -9765.679} C_VEL
LIN {X 0,Y 427.608,Z 280.824,A -85,B 0,C 180,E1 -9767.698,E2 -9767.698} C_VEL
LIN {X 0,Y 427.468,Z 285.511,A -85,B 0,C 180,E1 -9770.12,E2 -9770.12} C_VEL
LIN {X 0,Y 426.952,Z 291.625,A -85,B 0,C 180,E1 -9773.072,E2 -9773.072} C_VEL
LIN {X 0,Y 426.459,Z 299.114,A -85,B 0,C 180,E1 -9776.491,E2 -9776.491} C_VEL
LIN {X 0,Y 426.001,Z 306.678,A -85,B 0,C 180,E1 -9779.79,E2 -9779.79} C_VEL
LIN {X 0,Y 425.641,Z 314.543,A -85,B 0,C 180,E1 -9783.079,E2 -9783.079} C_VEL
LIN {X 0,Y 425.34,Z 321.501,A -85,B 0,C 180,E1 -9785.902,E2 -9785.902} C_VEL
LIN {X 0,Y 429.656,Z 339.805,A -85,B 0,C 180,E1 -9786.602,E2 -9786.602} C_VEL
LIN {X 0,Y 433.068,Z 355.219,A -85,B 0,C 180,E1 -9787.368,E2 -9787.368} C_VEL
LIN {X 0,Y 433.476,Z 358.454,A -85,B 0,C 180,E1 -9787.541,E2 -9787.541} C_VEL
LIN {X 0,Y 432.542,Z 373.454,A -85,B 0,C 180,E1 -9788.307,E2 -9788.307} C_VEL
LIN {X 0,Y 431.316,Z 387.847,A -85,B 0,C 180,E1 -9789.244,E2 -9789.244} C_VEL
LIN {X 0,Y 430.181,Z 400.99,A -85,B 0,C 180,E1 -9790.309,E2 -9790.309} C_VEL
LIN {X 0,Y 429.047,Z 413.144,A -85,B 0,C 180,E1 -9791.497,E2 -9791.497} C_VEL
LIN {X 0,Y 428.048,Z 424.423,A -85,B 0,C 180,E1 -9792.811,E2 -9792.811} C_VEL
LIN {X 0,Y 426.993,Z 434.796,A -85,B 0,C 180,E1 -9794.243,E2 -9794.243} C_VEL
LIN {X 0,Y 426.056,Z 444.963,A -85,B 0,C 180,E1 -9795.919,E2 -9795.919} C_VEL
LIN {X 0,Y 425.316,Z 454.527,A -85,B 0,C 180,E1 -9797.838,E2 -9797.838} C_VEL
LIN {X 0,Y 424.806,Z 461.373,A -85,B 0,C 180,E1 -9799.515,E2 -9799.515} C_VEL
LIN {X 0,Y 424.449,Z 467.71,A -85,B 0,C 180,E1 -9801.43,E2 -9801.43} C_VEL
LIN {X 0,Y 424.335,Z 473.189,A -85,B 0,C 180,E1 -9803.589,E2 -9803.589} C_VEL
LIN {X 0,Y 424.168,Z 476.218,A -85,B 0,C 180,E1 -9805.249,E2 -9805.249} C_VEL
LIN {X 0,Y 424.192,Z 478.596,A -85,B 0,C 180,E1 -9807.152,E2 -9807.152} C_VEL
LIN {X 0,Y 424.067,Z 479.789,A -85,B 0,C 180,E1 -9809.051,E2 -9809.051} C_VEL
LIN {X 0,Y 424.067,Z 479.799,A -85,B 0,C 180,E1 -9810.95,E2 -9810.95} C_VEL
LIN {X 0,Y 424.174,Z 478.62,A -85,B 0,C 180,E1 -9812.85,E2 -9812.85} C_VEL
LIN {X 0,Y 424.165,Z 476.264,A -85,B 0,C 180,E1 -9814.753,E2 -9814.753} C_VEL
LIN {X 0,Y 424.296,Z 472.695,A -85,B 0,C 180,E1 -9816.659,E2 -9816.659} C_VEL
LIN {X 0,Y 424.45,Z 467.815,A -85,B 0,C 180,E1 -9818.571,E2 -9818.571} C_VEL
LIN {X 0,Y 424.801,Z 461.503,A -85,B 0,C 180,E1 -9820.486,E2 -9820.486} C_VEL
LIN {X 0,Y 425.343,Z 454.691,A -85,B 0,C 180,E1 -9822.162,E2 -9822.162} C_VEL
LIN {X 0,Y 426.063,Z 445.173,A -85,B 0,C 180,E1 -9824.082,E2 -9824.082} C_VEL
LIN {X 0,Y 427.02,Z 435.053,A -85,B 0,C 180,E1 -9825.758,E2 -9825.758} C_VEL
LIN {X 0,Y 428.064,Z 424.725,A -85,B 0,C 180,E1 -9827.19,E2 -9827.19} C_VEL
LIN {X 0,Y 429.191,Z 412.416,A -85,B 0,C 180,E1 -9828.622,E2 -9828.622} C_VEL
LIN {X 0,Y 430.338,Z 400.086,A -85,B 0,C 180,E1 -9829.809,E2 -9829.809} C_VEL
LIN {X 0,Y 431.463,Z 386.682,A -85,B 0,C 180,E1 -9830.875,E2 -9830.875} C_VEL
LIN {X 0,Y 432.689,Z 371.926,A -85,B 0,C 180,E1 -9831.812,E2 -9831.812} C_VEL
LIN {X 0,Y 433.548,Z 357.646,A -85,B 0,C 180,E1 -9832.52,E2 -9832.52} C_VEL
LIN {X 0,Y 430.386,Z 343.113,A -85,B 0,C 180,E1 -9833.264,E2 -9833.264} C_VEL
LIN {X 0,Y 426.73,Z 327.785,A -85,B 0,C 180,E1 -9833.887,E2 -9833.887} C_VEL
LIN {X 0,Y 425.376,Z 322.221,A -85,B 0,C 180,E1 -9834.097,E2 -9834.097} C_VEL
LIN {X 0,Y 425.784,Z 313.877,A -85,B 0,C 180,E1 -9837.528,E2 -9837.528} C_VEL
LIN {X 0,Y 426.245,Z 305.765,A -85,B 0,C 180,E1 -9840.975,E2 -9840.975} C_VEL
LIN {X 0,Y 426.73,Z 297.626,A -85,B 0,C 180,E1 -9844.565,E2 -9844.565} C_VEL
LIN {X 0,Y 427.262,Z 290.517,A -85,B 0,C 180,E1 -9847.856,E2 -9847.856} C_VEL
LIN {X 0,Y 427.708,Z 284.218,A -85,B 0,C 180,E1 -9850.899,E2 -9850.899} C_VEL
LIN {X 0,Y 427.586,Z 280.145,A -85,B 0,C 180,E1 -9852.998,E2 -9852.998} C_VEL
LIN {X 0,Y 426.82,Z 275.333,A -85,B 0,C 180,E1 -9855.641,E2 -9855.641} C_VEL
LIN {X 0,Y 425.876,Z 270.16,A -85,B 0,C 180,E1 -9858.692,E2 -9858.692} C_VEL
LIN {X 0,Y 425.316,Z 267.133,A -85,B 0,C 180,E1 -9860.604,E2 -9860.604} C_VEL
LIN {X 0,Y 425.287,Z 267.135,A -85,B 0,C 180,E1 -9864.071,E2 -9864.071} C_VEL
LIN {X 0,Y 425.287,Z 267.137,A -85,B 0,C 180,E1 -9866.952,E2 -9866.952} C_VEL
LIN {X 0,Y 425.296,Z 267.134,A -85,B 0,C 180,E1 -9870.28,E2 -9870.28} C_VEL
LIN {X 0,Y 425.36,Z 267.124,A -85,B 0,C 180,E1 -9873.505,E2 -9873.505} C_VEL
LIN {X 0,Y 425.313,Z 267.134,A -85,B 0,C 180,E1 -9876.634,E2 -9876.634} C_VEL
LIN {X 0,Y 425.335,Z 267.13,A -85,B 0,C 180,E1 -9880.364,E2 -9880.364} C_VEL
LIN {X 0,Y 425.394,Z 267.12,A -85,B 0,C 180,E1 -9883.688,E2 -9883.688} C_VEL
LIN {X 0,Y 425.417,Z 267.117,A -85,B 0,C 180,E1 -9887.597,E2 -9887.597} C_VEL
LIN {X 0,Y 425.441,Z 267.113,A -85,B 0,C 180,E1 -9891.449,E2 -9891.449} C_VEL
LIN {X 0,Y 425.545,Z 267.105,A -85,B 0,C 180,E1 -9894.312,E2 -9894.312} C_VEL
LIN {X 0,Y 425.578,Z 267.099,A -85,B 0,C 180,E1 -9898.106,E2 -9898.106} C_VEL
LIN {X 0,Y 425.708,Z 267.083,A -85,B 0,C 180,E1 -9899.999,E2 -9899.999} C_VEL
LIN {X 0,Y 425.548,Z 267.103,A -85,B 0,C 180,E1 -9902.839,E2 -9902.839} C_VEL
LIN {X 0,Y 425.534,Z 267.105,A -85,B 0,C 180,E1 -9906.646,E2 -9906.646} C_VEL
LIN {X 0,Y 425.404,Z 267.118,A -85,B 0,C 180,E1 -9909.508,E2 -9909.508} C_VEL
LIN {X 0,Y 425.396,Z 267.12,A -85,B 0,C 180,E1 -9912.902,E2 -9912.902} C_VEL
LIN {X 0,Y 425.363,Z 267.126,A -85,B 0,C 180,E1 -9916.604,E2 -9916.604} C_VEL
LIN {X 0,Y 425.33,Z 267.129,A -85,B 0,C 180,E1 -9919.634,E2 -9919.634} C_VEL
LIN {X 0,Y 425.307,Z 267.131,A -85,B 0,C 180,E1 -9923.364,E2 -9923.364} C_VEL
LIN {X 0,Y 425.348,Z 267.126,A -85,B 0,C 180,E1 -9926.843,E2 -9926.843} C_VEL
LIN {X 0,Y 425.29,Z 267.136,A -85,B 0,C 180,E1 -9929.718,E2 -9929.718} C_VEL
LIN {X 0,Y 425.28,Z 267.133,A -85,B 0,C 180,E1 -9933.047,E2 -9933.047} C_VEL
LIN {X 0,Y 425.282,Z 267.138,A -85,B 0,C 180,E1 -9935.928,E2 -9935.928} C_VEL
LIN {X 0,Y 425.3,Z 267.131,A -85,B 0,C 180,E1 -9939.043,E2 -9939.043} C_VEL
LIN {X 0,Y 425.274,Z 267.135,A -85,B 0,C 180,E1 -9942.651,E2 -9942.651} C_VEL
LIN {X 0,Y 425.329,Z 267.131,A -85,B 0,C 180,E1 -9946.052,E2 -9946.052} C_VEL
LIN {X 0,Y 425.304,Z 267.13,A -85,B 0,C 180,E1 -9948.624,E2 -9948.624} C_VEL
LIN {X 0,Y 425.316,Z 267.13,A -85,B 0,C 180,E1 -9951.103,E2 -9951.103} C_VEL
LIN {X 0,Y 425.294,Z 267.132,A -85,B 0,C 180,E1 -9954.663,E2 -9954.663} C_VEL
LIN {X 0,Y 425.259,Z 267.139,A -85,B 0,C 180,E1 -9958.072,E2 -9958.072} C_VEL
LIN {X 0,Y 425.33,Z 267.131,A -85,B 0,C 180,E1 -9961.367,E2 -9961.367} C_VEL
LIN {X 0,Y 425.287,Z 267.132,A -85,B 0,C 180,E1 -9964.554,E2 -9964.554} C_VEL
LIN {X 0,Y 425.279,Z 267.138,A -85,B 0,C 180,E1 -9967.66,E2 -9967.66} C_VEL
LIN {X 0,Y 425.353,Z 267.125,A -85,B 0,C 180,E1 -9970.703,E2 -9970.703} C_VEL
LIN {X 0,Y 425.379,Z 267.125,A -85,B 0,C 180,E1 -9973.687,E2 -9973.687} C_VEL
LIN {X 0,Y 425.42,Z 267.12,A -85,B 0,C 180,E1 -9977.598,E2 -9977.598} C_VEL
LIN {X 0,Y 425.432,Z 267.119,A -85,B 0,C 180,E1 -9981.449,E2 -9981.449} C_VEL
LIN {X 0,Y 425.533,Z 267.102,A -85,B 0,C 180,E1 -9984.312,E2 -9984.312} C_VEL
LIN {X 0,Y 425.357,Z 267.332,A -85,B 0,C 180,E1 -9989.053,E2 -9989.053} C_VEL
LIN {X 0,Y 424.822,Z 271.518,A -85,B 0,C 180,E1 -9993.794,E2 -9993.794} C_VEL
LIN {X 0,Y 424.797,Z 274.348,A -85,B 0,C 180,E1 -9996.96,E2 -9996.96} C_VEL
LIN {X 0,Y 424.665,Z 276.252,A -85,B 0,C 180,E1 -9999.059,E2 -9999.059} C_VEL
LIN {X 0,Y 426.738,Z 277.905,A -85,B 0,C 180,E1 -9999.242,E2 -9999.242} C_VEL
LIN {X 0,Y 429.271,Z 281.618,A -85,B 0,C 180,E1 -9999.459,E2 -9999.459} C_VEL
LIN {X 0,Y 430.367,Z 285.363,A -85,B 0,C 180,E1 -9999.631,E2 -9999.631} C_VEL
LIN {X 0,Y 430.575,Z 289.585,A -85,B 0,C 180,E1 -9999.739,E2 -9999.739} C_VEL
LIN {X 0,Y 429.965,Z 293.133,A -85,B 0,C 180,E1 -9999.779,E2 -9999.779} C_VEL
LIN {X 0,Y 427.437,Z 301.055,A -85,B 0,C 180,E1 -9999.967,E2 -9999.967} C_VEL
LIN {X 0,Y 426.998,Z 304.384,A -85,B 0,C 180,E1 -10000.107,E2 -10000.107} C_VEL
LIN {X 0,Y 427.282,Z 306.519,A -85,B 0,C 180,E1 -10000.222,E2 -10000.222} C_VEL
LIN {X 0,Y 426.492,Z 321.112,A -85,B 0,C 180,E1 -10000.958,E2 -10000.958} C_VEL
LIN {X 0,Y 425.437,Z 335.861,A -85,B 0,C 180,E1 -10001.916,E2 -10001.916} C_VEL
LIN {X 0,Y 424.344,Z 349.264,A -85,B 0,C 180,E1 -10003.004,E2 -10003.004} C_VEL
LIN {X 0,Y 423.132,Z 362.337,A -85,B 0,C 180,E1 -10004.303,E2 -10004.303} C_VEL
LIN {X 0,Y 421.969,Z 373.998,A -85,B 0,C 180,E1 -10005.702,E2 -10005.702} C_VEL
LIN {X 0,Y 420.877,Z 384.699,A -85,B 0,C 180,E1 -10007.241,E2 -10007.241} C_VEL
LIN {X 0,Y 419.852,Z 393.784,A -85,B 0,C 180,E1 -10008.797,E2 -10008.797} C_VEL
LIN {X 0,Y 419.032,Z 402.609,A -85,B 0,C 180,E1 -10010.622,E2 -10010.622} C_VEL
LIN {X 0,Y 418.354,Z 409.996,A -85,B 0,C 180,E1 -10012.493,E2 -10012.493} C_VEL
LIN {X 0,Y 417.854,Z 415.615,A -85,B 0,C 180,E1 -10014.26,E2 -10014.26} C_VEL
LIN {X 0,Y 417.552,Z 419.92,A -85,B 0,C 180,E1 -10015.951,E2 -10015.951} C_VEL
LIN {X 0,Y 417.411,Z 422.162,A -85,B 0,C 180,E1 -10017.039,E2 -10017.039} C_VEL
LIN {X 0,Y 417.106,Z 425.545,A -85,B 0,C 180,E1 -10019.25,E2 -10019.25} C_VEL
LIN {X 0,Y 417.037,Z 426.991,A -85,B 0,C 180,E1 -10020.747,E2 -10020.747} C_VEL
LIN {X 0,Y 416.985,Z 427.794,A -85,B 0,C 180,E1 -10022.638,E2 -10022.638} C_VEL
LIN {X 0,Y 416.986,Z 427.638,A -85,B 0,C 180,E1 -10024.327,E2 -10024.327} C_VEL
LIN {X 0,Y 417.056,Z 426.499,A -85,B 0,C 180,E1 -10026.142,E2 -10026.142} C_VEL
LIN {X 0,Y 417.233,Z 424.748,A -85,B 0,C 180,E1 -10027.66,E2 -10027.66} C_VEL
LIN {X 0,Y 417.44,Z 422.161,A -85,B 0,C 180,E1 -10029.247,E2 -10029.247} C_VEL
LIN {X 0,Y 417.728,Z 418.302,A -85,B 0,C 180,E1 -10031.006,E2 -10031.006} C_VEL
LIN {X 0,Y 418.194,Z 412.967,A -85,B 0,C 180,E1 -10032.891,E2 -10032.891} C_VEL
LIN {X 0,Y 418.837,Z 406.105,A -85,B 0,C 180,E1 -10034.808,E2 -10034.808} C_VEL
LIN {X 0,Y 419.669,Z 397.995,A -85,B 0,C 180,E1 -10036.64,E2 -10036.64} C_VEL
LIN {X 0,Y 420.644,Z 388.92,A -85,B 0,C 180,E1 -10038.33,E2 -10038.33} C_VEL
LIN {X 0,Y 421.68,Z 379.129,A -85,B 0,C 180,E1 -10039.856,E2 -10039.856} C_VEL
LIN {X 0,Y 422.927,Z 367.561,A -85,B 0,C 180,E1 -10041.353,E2 -10041.353} C_VEL
LIN {X 0,Y 424.189,Z 355.19,A -85,B 0,C 180,E1 -10042.679,E2 -10042.679} C_VEL
LIN {X 0,Y 425.316,Z 342.579,A -85,B 0,C 180,E1 -10043.8,E2 -10043.8} C_VEL
LIN {X 0,Y 426.434,Z 329.084,A -85,B 0,C 180,E1 -10044.774,E2 -10044.774} C_VEL
LIN {X 0,Y 427.403,Z 314.246,A -85,B 0,C 180,E1 -10045.619,E2 -10045.619} C_VEL
LIN {X 0,Y 427.748,Z 308.28,A -85,B 0,C 180,E1 -10045.899,E2 -10045.899} C_VEL
LIN {X 0,Y 425.198,Z 299.106,A -85,B 0,C 180,E1 -10046.451,E2 -10046.451} C_VEL
LIN {X 0,Y 419.883,Z 284.205,A -85,B 0,C 180,E1 -10047.27,E2 -10047.27} C_VEL
LIN {X 0,Y 417.773,Z 278.593,A -85,B 0,C 180,E1 -10047.539,E2 -10047.539} C_VEL
LIN {X 0,Y 417.829,Z 275.567,A -85,B 0,C 180,E1 -10051.002,E2 -10051.002} C_VEL
LIN {X 0,Y 417.925,Z 273.09,A -85,B 0,C 180,E1 -10054.074,E2 -10054.074} C_VEL
LIN {X 0,Y 418.044,Z 270.574,A -85,B 0,C 180,E1 -10057.254,E2 -10057.254} C_VEL
LIN {X 0,Y 418.148,Z 268.149,A -85,B 0,C 180,E1 -10060.359,E2 -10060.359} C_VEL
LIN {X 0,Y 418.317,Z 268.009,A -85,B 0,C 180,E1 -10063.406,E2 -10063.406} C_VEL
LIN {X 0,Y 418.339,Z 268.001,A -85,B 0,C 180,E1 -10067,E2 -10067} C_VEL
LIN {X 0,Y 418.335,Z 268.003,A -85,B 0,C 180,E1 -10070.33,E2 -10070.33} C_VEL
LIN {X 0,Y 418.488,Z 267.984,A -85,B 0,C 180,E1 -10073.25,E2 -10073.25} C_VEL
LIN {X 0,Y 418.337,Z 268.003,A -85,B 0,C 180,E1 -10075.183,E2 -10075.183} C_VEL
LIN {X 0,Y 418.54,Z 267.975,A -85,B 0,C 180,E1 -10078.076,E2 -10078.076} C_VEL
LIN {X 0,Y 418.668,Z 267.958,A -85,B 0,C 180,E1 -10080.001,E2 -10080.001} C_VEL
LIN {X 0,Y 418.506,Z 267.981,A -85,B 0,C 180,E1 -10082.889,E2 -10082.889} C_VEL
LIN {X 0,Y 418.49,Z 267.982,A -85,B 0,C 180,E1 -10086.752,E2 -10086.752} C_VEL
LIN {X 0,Y 418.338,Z 268.002,A -85,B 0,C 180,E1 -10089.672,E2 -10089.672} C_VEL
LIN {X 0,Y 418.343,Z 267.998,A -85,B 0,C 180,E1 -10093.002,E2 -10093.002} C_VEL
LIN {X 0,Y 418.31,Z 268.003,A -85,B 0,C 180,E1 -10096.737,E2 -10096.737} C_VEL
LIN {X 0,Y 418.268,Z 268.009,A -85,B 0,C 180,E1 -10099.791,E2 -10099.791} C_VEL
LIN {X 0,Y 418.236,Z 268.015,A -85,B 0,C 180,E1 -10102.737,E2 -10102.737} C_VEL
LIN {X 0,Y 418.269,Z 268.011,A -85,B 0,C 180,E1 -10105.905,E2 -10105.905} C_VEL
LIN {X 0,Y 418.263,Z 268.012,A -85,B 0,C 180,E1 -10109.163,E2 -10109.163} C_VEL
LIN {X 0,Y 418.255,Z 268.018,A -85,B 0,C 180,E1 -10112.845,E2 -10112.845} C_VEL
LIN {X 0,Y 418.243,Z 268.021,A -85,B 0,C 180,E1 -10116.239,E2 -10116.239} C_VEL
LIN {X 0,Y 418.282,Z 268.138,A -85,B 0,C 180,E1 -10118.69,E2 -10118.69} C_VEL
LIN {X 0,Y 419.133,Z 272.976,A -85,B 0,C 180,E1 -10122.123,E2 -10122.123} C_VEL
LIN {X 0,Y 420.28,Z 279.151,A -85,B 0,C 180,E1 -10125.977,E2 -10125.977} C_VEL
LIN {X 0,Y 420.673,Z 282.863,A -85,B 0,C 180,E1 -10128.068,E2 -10128.068} C_VEL
LIN {X 0,Y 420.395,Z 287.672,A -85,B 0,C 180,E1 -10130.561,E2 -10130.561} C_VEL
LIN {X 0,Y 419.903,Z 293.6,A -85,B 0,C 180,E1 -10133.455,E2 -10133.455} C_VEL
LIN {X 0,Y 419.388,Z 301.052,A -85,B 0,C 180,E1 -10136.918,E2 -10136.918} C_VEL
LIN {X 0,Y 418.93,Z 308.751,A -85,B 0,C 180,E1 -10140.316,E2 -10140.316} C_VEL
LIN {X 0,Y 418.509,Z 316.456,A -85,B 0,C 180,E1 -10143.577,E2 -10143.577} C_VEL
LIN {X 0,Y 418.297,Z 320.994,A -85,B 0,C 180,E1 -10145.46,E2 -10145.46} C_VEL
LIN {X 0,Y 422.713,Z 339.468,A -85,B 0,C 180,E1 -10146.194,E2 -10146.194} C_VEL
LIN {X 0,Y 426.032,Z 354.599,A -85,B 0,C 180,E1 -10146.967,E2 -10146.967} C_VEL
LIN {X 0,Y 426.804,Z 359.403,A -85,B 0,C 180,E1 -10147.24,E2 -10147.24} C_VEL
LIN {X 0,Y 425.885,Z 372.972,A -85,B 0,C 180,E1 -10147.95,E2 -10147.95} C_VEL
LIN {X 0,Y 424.623,Z 387.361,A -85,B 0,C 180,E1 -10148.901,E2 -10148.901} C_VEL
LIN {X 0,Y 423.397,Z 400.497,A -85,B 0,C 180,E1 -10149.98,E2 -10149.98} C_VEL
LIN {X 0,Y 422.225,Z 412.651,A -85,B 0,C 180,E1 -10151.187,E2 -10151.187} C_VEL
LIN {X 0,Y 421.181,Z 423.932,A -85,B 0,C 180,E1 -10152.522,E2 -10152.522} C_VEL
LIN {X 0,Y 420.061,Z 434.308,A -85,B 0,C 180,E1 -10153.976,E2 -10153.976} C_VEL
LIN {X 0,Y 419.087,Z 444.483,A -85,B 0,C 180,E1 -10155.68,E2 -10155.68} C_VEL
LIN {X 0,Y 418.284,Z 454.055,A -85,B 0,C 180,E1 -10157.631,E2 -10157.631} C_VEL
LIN {X 0,Y 417.784,Z 460.909,A -85,B 0,C 180,E1 -10159.337,E2 -10159.337} C_VEL
LIN {X 0,Y 417.395,Z 467.252,A -85,B 0,C 180,E1 -10161.285,E2 -10161.285} C_VEL
LIN {X 0,Y 417.236,Z 472.169,A -85,B 0,C 180,E1 -10163.229,E2 -10163.229} C_VEL
LIN {X 0,Y 417.099,Z 475.773,A -85,B 0,C 180,E1 -10165.168,E2 -10165.168} C_VEL
LIN {X 0,Y 417.103,Z 478.153,A -85,B 0,C 180,E1 -10167.103,E2 -10167.103} C_VEL
LIN {X 0,Y 416.991,Z 479.352,A -85,B 0,C 180,E1 -10169.035,E2 -10169.035} C_VEL
LIN {X 0,Y 416.991,Z 479.365,A -85,B 0,C 180,E1 -10170.966,E2 -10170.966} C_VEL
LIN {X 0,Y 417.087,Z 478.188,A -85,B 0,C 180,E1 -10172.898,E2 -10172.898} C_VEL
LIN {X 0,Y 417.095,Z 475.833,A -85,B 0,C 180,E1 -10174.834,E2 -10174.834} C_VEL
LIN {X 0,Y 417.228,Z 472.263,A -85,B 0,C 180,E1 -10176.772,E2 -10176.772} C_VEL
LIN {X 0,Y 417.396,Z 467.383,A -85,B 0,C 180,E1 -10178.717,E2 -10178.717} C_VEL
LIN {X 0,Y 417.78,Z 461.07,A -85,B 0,C 180,E1 -10180.664,E2 -10180.664} C_VEL
LIN {X 0,Y 418.317,Z 454.257,A -85,B 0,C 180,E1 -10182.37,E2 -10182.37} C_VEL
LIN {X 0,Y 419.092,Z 444.737,A -85,B 0,C 180,E1 -10184.321,E2 -10184.321} C_VEL
LIN {X 0,Y 420.093,Z 434.616,A -85,B 0,C 180,E1 -10186.025,E2 -10186.025} C_VEL
LIN {X 0,Y 421.206,Z 424.29,A -85,B 0,C 180,E1 -10187.478,E2 -10187.478} C_VEL
LIN {X 0,Y 422.372,Z 411.979,A -85,B 0,C 180,E1 -10188.934,E2 -10188.934} C_VEL
LIN {X 0,Y 423.58,Z 399.651,A -85,B 0,C 180,E1 -10190.139,E2 -10190.139} C_VEL
LIN {X 0,Y 424.774,Z 386.249,A -85,B 0,C 180,E1 -10191.219,E2 -10191.219} C_VEL
LIN {X 0,Y 426.069,Z 371.493,A -85,B 0,C 180,E1 -10192.169,E2 -10192.169} C_VEL
LIN {X 0,Y 426.879,Z 359.394,A -85,B 0,C 180,E1 -10192.784,E2 -10192.784} C_VEL
LIN {X 0,Y 423.958,Z 345.269,A -85,B 0,C 180,E1 -10193.545,E2 -10193.545} C_VEL
LIN {X 0,Y 420.432,Z 330.084,A -85,B 0,C 180,E1 -10194.207,E2 -10194.207} C_VEL
LIN {X 0,Y 418.343,Z 321.832,A -85,B 0,C 180,E1 -10194.514,E2 -10194.514} C_VEL
LIN {X 0,Y 418.781,Z 313.481,A -85,B 0,C 180,E1 -10198.028,E2 -10198.028} C_VEL
LIN {X 0,Y 419.22,Z 306.096,A -85,B 0,C 180,E1 -10201.241,E2 -10201.241} C_VEL
LIN {X 0,Y 419.733,Z 298.076,A -85,B 0,C 180,E1 -10204.869,E2 -10204.869} C_VEL
LIN {X 0,Y 420.315,Z 290.958,A -85,B 0,C 180,E1 -10208.22,E2 -10208.22} C_VEL
LIN {X 0,Y 420.704,Z 285.98,A -85,B 0,C 180,E1 -10210.656,E2 -10210.656} C_VEL
LIN {X 0,Y 420.67,Z 282.089,A -85,B 0,C 180,E1 -10212.684,E2 -10212.684} C_VEL
LIN {X 0,Y 419.957,Z 277.297,A -85,B 0,C 180,E1 -10215.341,E2 -10215.341} C_VEL
LIN {X 0,Y 418.854,Z 271.11,A -85,B 0,C 180,E1 -10219.031,E2 -10219.031} C_VEL
LIN {X 0,Y 418.264,Z 268.011,A -85,B 0,C 180,E1 -10221.071,E2 -10221.071} C_VEL
LIN {X 0,Y 418.248,Z 268.012,A -85,B 0,C 180,E1 -10223.976,E2 -10223.976} C_VEL
LIN {X 0,Y 418.263,Z 268.011,A -85,B 0,C 180,E1 -10227.156,E2 -10227.156} C_VEL
LIN {X 0,Y 418.274,Z 268.011,A -85,B 0,C 180,E1 -10230.895,E2 -10230.895} C_VEL
LIN {X 0,Y 418.277,Z 268.007,A -85,B 0,C 180,E1 -10234.096,E2 -10234.096} C_VEL
LIN {X 0,Y 418.244,Z 268.011,A -85,B 0,C 180,E1 -10237.263,E2 -10237.263} C_VEL
LIN {X 0,Y 418.289,Z 268.007,A -85,B 0,C 180,E1 -10240.364,E2 -10240.364} C_VEL
LIN {X 0,Y 418.323,Z 268,A -85,B 0,C 180,E1 -10243.404,E2 -10243.404} C_VEL
LIN {X 0,Y 418.352,Z 267.999,A -85,B 0,C 180,E1 -10246.999,E2 -10246.999} C_VEL
LIN {X 0,Y 418.345,Z 268.001,A -85,B 0,C 180,E1 -10250.328,E2 -10250.328} C_VEL
LIN {X 0,Y 418.464,Z 267.983,A -85,B 0,C 180,E1 -10253.248,E2 -10253.248} C_VEL
LIN {X 0,Y 418.34,Z 267.998,A -85,B 0,C 180,E1 -10255.181,E2 -10255.181} C_VEL
LIN {X 0,Y 418.547,Z 267.975,A -85,B 0,C 180,E1 -10258.074,E2 -10258.074} C_VEL
LIN {X 0,Y 418.677,Z 267.958,A -85,B 0,C 180,E1 -10259.999,E2 -10259.999} C_VEL
LIN {X 0,Y 418.504,Z 267.98,A -85,B 0,C 180,E1 -10262.887,E2 -10262.887} C_VEL
LIN {X 0,Y 418.497,Z 267.981,A -85,B 0,C 180,E1 -10266.75,E2 -10266.75} C_VEL
LIN {X 0,Y 418.403,Z 267.993,A -85,B 0,C 180,E1 -10268.694,E2 -10268.694} C_VEL
LIN {X 0,Y 418.318,Z 268.001,A -85,B 0,C 180,E1 -10271.63,E2 -10271.63} C_VEL
LIN {X 0,Y 418.305,Z 268.005,A -85,B 0,C 180,E1 -10274.596,E2 -10274.596} C_VEL
LIN {X 0,Y 418.29,Z 268.005,A -85,B 0,C 180,E1 -10277.602,E2 -10277.602} C_VEL
LIN {X 0,Y 418.251,Z 268.011,A -85,B 0,C 180,E1 -10280.662,E2 -10280.662} C_VEL
LIN {X 0,Y 418.288,Z 268.008,A -85,B 0,C 180,E1 -10283.78,E2 -10283.78} C_VEL
LIN {X 0,Y 418.309,Z 268.002,A -85,B 0,C 180,E1 -10287.069,E2 -10287.069} C_VEL
LIN {X 0,Y 418.243,Z 268.014,A -85,B 0,C 180,E1 -10290.271,E2 -10290.271} C_VEL
LIN {X 0,Y 418.247,Z 268.013,A -85,B 0,C 180,E1 -10293.676,E2 -10293.676} C_VEL
LIN {X 0,Y 418.243,Z 268.011,A -85,B 0,C 180,E1 -10297.222,E2 -10297.222} C_VEL
LIN {X 0,Y 418.252,Z 268.013,A -85,B 0,C 180,E1 -10299.68,E2 -10299.68} C_VEL
LIN {X 0,Y 418.228,Z 268.014,A -85,B 0,C 180,E1 -10302.32,E2 -10302.32} C_VEL
LIN {X 0,Y 418.256,Z 268.009,A -85,B 0,C 180,E1 -10305.111,E2 -10305.111} C_VEL
LIN {X 0,Y 418.287,Z 268.009,A -85,B 0,C 180,E1 -10307.772,E2 -10307.772} C_VEL
LIN {X 0,Y 418.259,Z 268.012,A -85,B 0,C 180,E1 -10311.558,E2 -10311.558} C_VEL
LIN {X 0,Y 418.253,Z 268.01,A -85,B 0,C 180,E1 -10315.158,E2 -10315.158} C_VEL
LIN {X 0,Y 418.238,Z 268.015,A -85,B 0,C 180,E1 -10317.471,E2 -10317.471} C_VEL
LIN {X 0,Y 418.269,Z 268.007,A -85,B 0,C 180,E1 -10320.892,E2 -10320.892} C_VEL
LIN {X 0,Y 418.263,Z 268.009,A -85,B 0,C 180,E1 -10324.095,E2 -10324.095} C_VEL
LIN {X 0,Y 418.229,Z 268.015,A -85,B 0,C 180,E1 -10327.263,E2 -10327.263} C_VEL
LIN {X 0,Y 418.274,Z 268.006,A -85,B 0,C 180,E1 -10330.363,E2 -10330.363} C_VEL
LIN {X 0,Y 418.307,Z 268.007,A -85,B 0,C 180,E1 -10333.404,E2 -10333.404} C_VEL
LIN {X 0,Y 418.345,Z 268,A -85,B 0,C 180,E1 -10336.993,E2 -10336.993} C_VEL
LIN {X 0,Y 418.351,Z 267.996,A -85,B 0,C 180,E1 -10340.328,E2 -10340.328} C_VEL
LIN {X 0,Y 418.48,Z 267.985,A -85,B 0,C 180,E1 -10343.248,E2 -10343.248} C_VEL
LIN {X 0,Y 418.276,Z 268.011,A -85,B 0,C 180,E1 -10345.18,E2 -10345.18} C_VEL
LIN {X 0,Y 418.324,Z 268.167,A -85,B 0,C 180,E1 -10349.037,E2 -10349.037} C_VEL
